            IF rtb_Divide_h >= 0.5 THEN 
                rtb_Add_d := rt_floorf(u := rtb_Add_d + 0.5);
            ELSE 
                rtb_Add_d := 0.0;
            END_IF;

        END_IF;

        (* Outputs for Atomic SubSystem: '<S676>/BatteryPackSignals' *)
        (* Product: '<S951>/Divide' incorporates:
         *  Constant: '<S811>/Constant8'
         *  SignalConversion: '<S682>/BusConversion_InsertedFor_IT_BatterySignal_Databus_at_inport_0' *)
        rtb_Add_en := rtb_Add_en / 100.0;
        (* End of Outputs for SubSystem: '<S676>/BatteryPackSignals' *)
        

        (* DataTypeConversion: '<S947>/Data Type Conversion2' *)
        rtb_Divide_h := ABS(rtb_Add_en);

        IF rtb_Divide_h < 8.388608E+6 THEN 

            IF rtb_Divide_h >= 0.5 THEN 
                rtb_Add_en := rt_floorf(u := rtb_Add_en + 0.5);
            ELSE 
                rtb_Add_en := 0.0;
            END_IF;

        END_IF;

        (* Outputs for Atomic SubSystem: '<S676>/BatteryPackSignals' *)
        (* Product: '<S964>/Divide' incorporates:
         *  Constant: '<S812>/Constant6'
         *  SignalConversion: '<S682>/BusConversion_InsertedFor_IT_BatterySignal_Databus_at_inport_0' *)
        rtb_Divide_h := rtb_Add_cw / 0.1;
        (* End of Outputs for SubSystem: '<S676>/BatteryPackSignals' *)
        

        (* DataTypeConversion: '<S960>/Data Type Conversion2' *)

        IF rtb_Divide_h >= 0.5 THEN 
            rtb_Add_ky := rt_floorf(u := rtb_Divide_h + 0.5);
        ELSE 
            rtb_Add_ky := 0.0;
        END_IF;

        (* Outputs for Atomic SubSystem: '<S676>/BatteryPackSignals' *)
        (* Product: '<S965>/Divide' incorporates:
         *  Constant: '<S812>/Constant8'
         *  SignalConversion: '<S682>/BusConversion_InsertedFor_IT_BatterySignal_Databus_at_inport_0' *)
        rtb_Divide_h := rtb_Add_bh / 0.1;
        (* End of Outputs for SubSystem: '<S676>/BatteryPackSignals' *)
        

        (* DataTypeConversion: '<S961>/Data Type Conversion2' *)

        IF rtb_Divide_h >= 0.5 THEN 
            rtb_Add_bh := rt_floorf(u := rtb_Divide_h + 0.5);
        ELSE 
            rtb_Add_bh := 0.0;
        END_IF;

        (* DataTypeConversion: '<S973>/Data Type Conversion4' *)
        v := ABS(rtb_BattSelect_i);

        IF v < 4.503599627370496E+15 THEN 

            IF v >= 0.5 THEN 
                rtb_BattSelect_i := rt_floord(u := rtb_BattSelect_i + 0.5);
            ELSE 
                rtb_BattSelect_i := 0.0;
            END_IF;

        END_IF;

        (* DataTypeConversion: '<S973>/Data Type Conversion1' *)
        v := ABS(rtb_BattSelect);

        IF v < 4.503599627370496E+15 THEN 

            IF v >= 0.5 THEN 
                rtb_BattSelect := rt_floord(u := rtb_BattSelect + 0.5);
            ELSE 
                rtb_BattSelect := 0.0;
            END_IF;

        END_IF;

        (* DataTypeConversion: '<S973>/Data Type Conversion3' *)
        v := ABS(rtb_BattSelect_f);

        IF v < 4.503599627370496E+15 THEN 

            IF v >= 0.5 THEN 
                rtb_BattSelect_f := rt_floord(u := rtb_BattSelect_f + 0.5);
            ELSE 
                rtb_BattSelect_f := 0.0;
            END_IF;

        END_IF;

        (* Outport: '<Root>/OP_ChiefMaster_IP_Msg1' incorporates:
         *  ArithShift: '<S973>/Shift Arithmetic1'
         *  ArithShift: '<S973>/Shift Arithmetic3'
         *  ArithShift: '<S973>/Shift Arithmetic5'
         *  ArithShift: '<S973>/Shift Arithmetic6'
         *  DataTypeConversion: '<S973>/Data Type Conversion1'
         *  DataTypeConversion: '<S973>/Data Type Conversion3'
         *  DataTypeConversion: '<S973>/Data Type Conversion4'
         *  DataTypeConversion: '<S973>/Data Type Conversion6'
         *  DataTypeConversion: '<S973>/Data Type Conversion7'
         *  SignalConversion: '<S677>/Signal Copy14'
         *  Sum: '<S973>/Add' *)
        OP_ChiefMaster_IP_Msg1[2] := UDINT_TO_USINT(USINT_TO_UDINT(UDINT_TO_USINT(USINT_TO_UDINT(UDINT_TO_USINT(USINT_TO_UDINT(UDINT_TO_USINT(USINT_TO_UDINT(UDINT_TO_USINT(USINT_TO_UDINT(UDINT_TO_USINT((DINT_TO_UDINT(DWORD_TO_DINT(SHL(DINT_TO_DWORD(BOOL_TO_DINT(DI_HVIL_Overrule)), 7))) + DINT_TO_UDINT(DWORD_TO_DINT(SHL(DINT_TO_DWORD(BOOL_TO_DINT(rtb_IT_boUDC_SafeToShutdown)), 6)))) + USINT_TO_UDINT(ShiftArithmetic4_m))) + USINT_TO_UDINT(BYTE_TO_USINT(SHL(USINT_TO_BYTE(DINT_TO_USINT(TRUNC(rtb_BattSelect_i))), 4))))) + USINT_TO_UDINT(ShiftArithmetic2_k))) + USINT_TO_UDINT(BYTE_TO_USINT(SHL(USINT_TO_BYTE(DINT_TO_USINT(TRUNC(rtb_BattSelect))), 2))))) + USINT_TO_UDINT(ShiftArithmetic_m))) + USINT_TO_UDINT(DINT_TO_USINT(TRUNC(rtb_BattSelect_f))));
        (* Product: '<S978>/Divide' incorporates:
         *  Constant: '<S976>/Constant2'
         *  Sum: '<S978>/Add' *)
        rtb_Divide_h := DINT_TO_REAL(rtb_Add_kr) / 0.1;
        (* DataTypeConversion: '<S977>/Data Type Conversion2' *)

        IF rtb_Divide_h >= 0.5 THEN 
            y_1 := rt_floorf(u := rtb_Divide_h + 0.5);
        ELSE 
            y_1 := 0.0;
        END_IF;

        (* DataTypeConversion: '<S981>/Data Type Conversion2' *)

        IF v_tmp < 4.503599627370496E+15 THEN 

            IF v_tmp >= 0.5 THEN 
                Count_k := rt_floord(u := REQ_HV_ON + 0.5);
            ELSE 
                Count_k := 0.0;
            END_IF;

        ELSE 
            Count_k := REQ_HV_ON;
        END_IF;

        (* DataTypeConversion: '<S981>/Data Type Conversion1' *)

        IF rtb_UnitDelay2 < 4.503599627370496E+15 THEN 

            IF rtb_UnitDelay2 >= 0.5 THEN 
                y := rt_floord(u := REQ_HV_ON_d + 0.5);
            ELSE 
                y := 0.0;
            END_IF;

        ELSE 
            y := REQ_HV_ON_d;
        END_IF;

        (* DataTypeConversion: '<S981>/Data Type Conversion' *)

        IF rtb_Uk1 < 4.503599627370496E+15 THEN 

            IF rtb_Uk1 >= 0.5 THEN 
                v := rt_floord(u := REQ_HV_ON_a + 0.5);
            ELSE 
                v := 0.0;
            END_IF;

        ELSE 
            v := REQ_HV_ON_a;
        END_IF;

        (* Outport: '<Root>/OP_ChiefMaster_OP_Msg2' incorporates:
         *  ArithShift: '<S981>/Shift Arithmetic'
         *  ArithShift: '<S981>/Shift Arithmetic1'
         *  ArithShift: '<S981>/Shift Arithmetic2'
         *  ArithShift: '<S981>/Shift Arithmetic3'
         *  ArithShift: '<S981>/Shift Arithmetic4'
         *  ArithShift: '<S982>/Shift Arithmetic'
         *  ArithShift: '<S982>/Shift Arithmetic1'
         *  DataTypeConversion: '<S981>/Data Type Conversion'
         *  DataTypeConversion: '<S981>/Data Type Conversion1'
         *  DataTypeConversion: '<S981>/Data Type Conversion2'
         *  DataTypeConversion: '<S981>/Data Type Conversion3'
         *  DataTypeConversion: '<S981>/Data Type Conversion4'
         *  DataTypeConversion: '<S981>/Data Type Conversion5'
         *  DataTypeConversion: '<S982>/Data Type Conversion'
         *  DataTypeConversion: '<S982>/Data Type Conversion1'
         *  DataTypeConversion: '<S982>/Data Type Conversion3'
         *  Outport: '<Root>/DO_boEMSRET_BB1_1'
         *  Sum: '<S981>/Add'
         *  Sum: '<S982>/Add' *)
        OP_ChiefMaster_OP_Msg2[1] := UDINT_TO_USINT(USINT_TO_UDINT(UDINT_TO_USINT(USINT_TO_UDINT(UDINT_TO_USINT(USINT_TO_UDINT(UDINT_TO_USINT(USINT_TO_UDINT(UDINT_TO_USINT(USINT_TO_UDINT(UDINT_TO_USINT(USINT_TO_UDINT(UDINT_TO_USINT(USINT_TO_UDINT(ShiftArithmetic6_i) + USINT_TO_UDINT(ShiftArithmetic5_k))) + DINT_TO_UDINT(DWORD_TO_DINT(SHL(DINT_TO_DWORD(BOOL_TO_DINT(DO_REQ_DC_ON_PLUS)), 5))))) + DINT_TO_UDINT(DWORD_TO_DINT(SHL(DINT_TO_DWORD(BOOL_TO_DINT(DO_REQ_DC_ON_MINUS)), 4))))) + USINT_TO_UDINT(BYTE_TO_USINT(SHL(USINT_TO_BYTE(DINT_TO_USINT(TRUNC(Count_k))), 3))))) + USINT_TO_UDINT(BYTE_TO_USINT(SHL(USINT_TO_BYTE(DINT_TO_USINT(TRUNC(y))), 2))))) + USINT_TO_UDINT(BYTE_TO_USINT(SHL(USINT_TO_BYTE(DINT_TO_USINT(TRUNC(v))), 1))))) + BOOL_TO_UDINT(DO_boKL15_IMD_BB3));
        OP_ChiefMaster_OP_Msg2[2] := UDINT_TO_USINT(USINT_TO_UDINT(UDINT_TO_USINT(USINT_TO_UDINT(UDINT_TO_USINT(USINT_TO_UDINT(UDINT_TO_USINT(USINT_TO_UDINT(UDINT_TO_USINT(USINT_TO_UDINT(UDINT_TO_USINT(USINT_TO_UDINT(UDINT_TO_USINT(USINT_TO_UDINT(ShiftArithmetic6_m) + USINT_TO_UDINT(ShiftArithmetic5_a))) + USINT_TO_UDINT(ShiftArithmetic4_a))) + USINT_TO_UDINT(ShiftArithmetic3_k))) + USINT_TO_UDINT(ShiftArithmetic2_p))) + DINT_TO_UDINT(DWORD_TO_DINT(SHL(DINT_TO_DWORD(BOOL_TO_DINT(DO_boResetButton_LED)), 2))))) + DINT_TO_UDINT(DWORD_TO_DINT(SHL(DINT_TO_DWORD(BOOL_TO_DINT(DO_boEMSRET_BB1_1)), 1))))) + BOOL_TO_UDINT(DO_CabinAlarm));
        (* ArithShift: '<S990>/Shift Arithmetic3' incorporates:
         *  DataTypeConversion: '<S990>/Data Type Conversion4' *)
        rtb_ShiftArithmetic3_p := DINT_TO_USINT(DWORD_TO_DINT(SHL(DINT_TO_DWORD(BOOL_TO_DINT(System_Error)), 4)));
        (* Outport: '<Root>/OP_ChiefMaster_SS1_Msg3' incorporates:
         *  ArithShift: '<S991>/Shift Arithmetic'
         *  ArithShift: '<S991>/Shift Arithmetic1'
         *  ArithShift: '<S991>/Shift Arithmetic3'
         *  ArithShift: '<S991>/Shift Arithmetic5'
         *  DataTypeConversion: '<S984>/Extract Desired Bits'
         *  DataTypeConversion: '<S985>/Extract Desired Bits'
         *  DataTypeConversion: '<S991>/Data Type Conversion'
         *  DataTypeConversion: '<S991>/Data Type Conversion3'
         *  Sum: '<S991>/Add' *)
        OP_ChiefMaster_SS1_Msg3[1] := UDINT_TO_USINT(USINT_TO_UDINT(UDINT_TO_USINT(USINT_TO_UDINT(UDINT_TO_USINT(USINT_TO_UDINT(UDINT_TO_USINT(USINT_TO_UDINT(UDINT_TO_USINT(USINT_TO_UDINT(UDINT_TO_USINT(USINT_TO_UDINT(UDINT_TO_USINT(DINT_TO_UDINT(DWORD_TO_DINT(SHL(DINT_TO_DWORD(USINT_TO_DINT(rtb_Out)) AND 3, 6))) + USINT_TO_UDINT(ShiftArithmetic6_h))) + USINT_TO_UDINT(ShiftArithmetic4_n))) + DINT_TO_UDINT(DWORD_TO_DINT(SHL(DINT_TO_DWORD(USINT_TO_DINT(rtb_ExtractDesiredBits_bk_tmp)), 4))))) + USINT_TO_UDINT(ShiftArithmetic2_d))) + DINT_TO_UDINT(DWORD_TO_DINT(SHL(DINT_TO_DWORD(USINT_TO_DINT(rtb_ExtractDesiredBits_b13)), 2))))) + DINT_TO_UDINT(DWORD_TO_DINT(SHL(DINT_TO_DWORD(BOOL_TO_DINT(rtb_IT_boBMS_HV_ON_BB)), 1))))) + BOOL_TO_UDINT(rtb_FL_boKL15_Reset));
        (* Outputs for Atomic SubSystem: '<S676>/BatteryPackSignals' *)
        (* Switch: '<S995>/Switch' incorporates:
         *  Constant: '<S994>/Constant2'
         *  SignalConversion: '<S682>/BusConversion_InsertedFor_IT_BatterySignal_Databus_at_inport_0' *)

        IF rtb_IP_boBMS_HV_REL_ON_BB1 THEN 
            rtb_Divide_h := rtb_Add_nm;
        ELSE 
            rtb_Divide_h := FL_sHVC_CellBalanceVoltage_mV;
        END_IF;

        (* End of Switch: '<S995>/Switch' *)
        (* End of Outputs for SubSystem: '<S676>/BatteryPackSignals' *)
        

        (* RelationalOperator: '<S996>/Relational Operator' incorporates:
         *  Constant: '<S994>/Constant2' *)
        rtb_boData_Out := rtb_Divide_h >= FL_sHVC_CellBalanceVoltage_mV;
        (* Outputs for Atomic SubSystem: '<S676>/BatteryPackSignals' *)
        (* Switch: '<S995>/Switch1' incorporates:
         *  Constant: '<S994>/Constant2'
         *  SignalConversion: '<S682>/BusConversion_InsertedFor_IT_BatterySignal_Databus_at_inport_0' *)

        IF rtb_IP_boBMS_HV_REL_ON_BB2 THEN 
            rtb_Divide_h := rtb_Add_d4;
        ELSE 
            rtb_Divide_h := FL_sHVC_CellBalanceVoltage_mV;
        END_IF;

        (* End of Switch: '<S995>/Switch1' *)
        (* End of Outputs for SubSystem: '<S676>/BatteryPackSignals' *)
        

        (* RelationalOperator: '<S996>/Relational Operator1' incorporates:
         *  Constant: '<S994>/Constant2' *)
        rtb_IT_boBMS_HV_ON_BB := rtb_Divide_h >= FL_sHVC_CellBalanceVoltage_mV;
        (* Outputs for Atomic SubSystem: '<S676>/BatteryPackSignals' *)
        (* Switch: '<S995>/Switch2' incorporates:
         *  Constant: '<S994>/Constant2'
         *  SignalConversion: '<S682>/BusConversion_InsertedFor_IT_BatterySignal_Databus_at_inport_0' *)

        IF rtb_IP_boBMS_HV_REL_ON_BB3 THEN 
            rtb_Divide_h := rtb_Add_cw;
        ELSE 
            rtb_Divide_h := FL_sHVC_CellBalanceVoltage_mV;
        END_IF;

        (* End of Switch: '<S995>/Switch2' *)
        (* End of Outputs for SubSystem: '<S676>/BatteryPackSignals' *)
        

        (* Outport: '<Root>/OP_ChiefMaster_SS1_Msg3' incorporates:
         *  ArithShift: '<S992>/Shift Arithmetic'
         *  ArithShift: '<S992>/Shift Arithmetic1'
         *  ArithShift: '<S992>/Shift Arithmetic4'
         *  ArithShift: '<S993>/Shift Arithmetic2'
         *  Constant: '<S994>/Constant2'
         *  DataTypeConversion: '<S987>/Extract Desired Bits'
         *  DataTypeConversion: '<S988>/Extract Desired Bits'
         *  DataTypeConversion: '<S989>/Extract Desired Bits'
         *  DataTypeConversion: '<S992>/Data Type Conversion'
         *  DataTypeConversion: '<S992>/Data Type Conversion1'
         *  DataTypeConversion: '<S992>/Data Type Conversion3'
         *  Logic: '<S996>/OR'
         *  RelationalOperator: '<S996>/Relational Operator2'
         *  Sum: '<S992>/Add'
         *  Sum: '<S993>/Add' *)
        OP_ChiefMaster_SS1_Msg3[2] := UDINT_TO_USINT(USINT_TO_UDINT(UDINT_TO_USINT(USINT_TO_UDINT(UDINT_TO_USINT(USINT_TO_UDINT(UDINT_TO_USINT(USINT_TO_UDINT(UDINT_TO_USINT(USINT_TO_UDINT(UDINT_TO_USINT(DINT_TO_UDINT(DWORD_TO_DINT(SHL(DINT_TO_DWORD(USINT_TO_DINT(rtb_IMD_State_g)) AND 7, 5))) + USINT_TO_UDINT(UDINT_TO_USINT(USINT_TO_UDINT(ShiftArithmetic6_n) + USINT_TO_UDINT(ShiftArithmetic5_a2))))) + USINT_TO_UDINT(ShiftArithmetic3_o))) + USINT_TO_UDINT(ShiftArithmetic2_b))) + DINT_TO_UDINT(DWORD_TO_DINT(SHL(DINT_TO_DWORD(BOOL_TO_DINT((rtb_boData_Out AND rtb_IT_boBMS_HV_ON_BB) AND (rtb_Divide_h >= FL_sHVC_CellBalanceVoltage_mV))), 2))))) + DINT_TO_UDINT(DWORD_TO_DINT(SHL(DINT_TO_DWORD(BOOL_TO_DINT(rtb_FL_boSS_HVIL_NOK)), 1))))) + BOOL_TO_UDINT(rtb_FL_boCMSleep));
        OP_ChiefMaster_SS1_Msg3[7] := UDINT_TO_USINT(USINT_TO_UDINT(UDINT_TO_USINT(USINT_TO_UDINT(UDINT_TO_USINT(USINT_TO_UDINT(UDINT_TO_USINT(USINT_TO_UDINT(UDINT_TO_USINT(USINT_TO_UDINT(UDINT_TO_USINT(USINT_TO_UDINT(UDINT_TO_USINT(USINT_TO_UDINT(ShiftArithmetic6_k) + USINT_TO_UDINT(ShiftArithmetic5_i))) + USINT_TO_UDINT(ShiftArithmetic4_ap))) + USINT_TO_UDINT(ShiftArithmetic3_e))) + DINT_TO_UDINT(DWORD_TO_DINT(SHL(DINT_TO_DWORD(USINT_TO_DINT(rtb_IMD_State)) AND 7, 3))))) + USINT_TO_UDINT(ShiftArithmetic1))) + USINT_TO_UDINT(ShiftArithmetic_h))) + DINT_TO_UDINT(DWORD_TO_DINT(DINT_TO_DWORD(USINT_TO_DINT(rtb_System_SD_ErrorCode)) AND 7)));
        (* Outputs for Atomic SubSystem: '<S676>/BatteryPackSignals' *)
        (* Product: '<S1002>/Divide' incorporates:
         *  Constant: '<S997>/Constant1'
         *  SignalConversion: '<S682>/BusConversion_InsertedFor_IT_BatterySignal_Databus_at_inport_0'
         *  Sum: '<S119>/Add' *)
        rtb_Divide_h := ((rtb_Add_ki5 + rtb_Add_ir) + rtb_Add_m) / 0.1;
        (* End of Outputs for SubSystem: '<S676>/BatteryPackSignals' *)
        

        (* DataTypeConversion: '<S1001>/Data Type Conversion2' *)

        IF ABS(rtb_Divide_h) >= 0.5 THEN 
            rtb_Add_nm := rt_floorf(u := rtb_Divide_h + 0.5);
        ELSE 
            rtb_Add_nm := 0.0;
        END_IF;

        (* DataTypeConversion: '<S1005>/Data Type Conversion2' incorporates:
         *  MinMax: '<S120>/Min' *)

        IF maxV >= 0.5 THEN 
            maxV := rt_floorf(u := maxV + 0.5);
        ELSE 
            maxV := 0.0;
        END_IF;

        (* DataTypeConversion: '<S1009>/Data Type Conversion2' incorporates:
         *  Sum: '<S1010>/Add' *)
        rtb_Divide_h := ABS(FL_sST_MaxChargeCurrent);

        IF rtb_Divide_h < 8.388608E+6 THEN 

            IF rtb_Divide_h >= 0.5 THEN 
                rtb_Add_d4 := rt_floorf(u := FL_sST_MaxChargeCurrent + 0.5);
            ELSE 
                rtb_Add_d4 := 0.0;
            END_IF;

        ELSE 
            rtb_Add_d4 := FL_sST_MaxChargeCurrent;
        END_IF;

        (* DataTypeConversion: '<S1013>/Data Type Conversion2' incorporates:
         *  Sum: '<S1014>/Add' *)
        rtb_Divide_h := ABS(rtb_FL_sSS_MaxDisChargeCurrent);

        IF rtb_Divide_h < 8.388608E+6 THEN 

            IF rtb_Divide_h >= 0.5 THEN 
                rtb_FL_sSS_MaxDisChargeCurrent := rt_floorf(u := rtb_FL_sSS_MaxDisChargeCurrent + 0.5);
            ELSE 
                rtb_FL_sSS_MaxDisChargeCurrent := 0.0;
            END_IF;

        END_IF;

        (* DataTypeConversion: '<S1020>/Data Type Conversion3' *)

        IF rtb_Uk1 < 4.503599627370496E+15 THEN 

            IF rtb_Uk1 >= 0.5 THEN 
                Count_k := rt_floord(u := REQ_HV_ON_a + 0.5);
            ELSE 
                Count_k := 0.0;
            END_IF;

        ELSE 
            Count_k := REQ_HV_ON_a;
        END_IF;

        (* Outport: '<Root>/BMS_Control_Batt1' incorporates:
         *  DataTypeConversion: '<S1020>/Data Type Conversion3'
         *  Sum: '<S1020>/Add' *)
        BMS_Control_Batt1[0] := UDINT_TO_USINT(USINT_TO_UDINT(UDINT_TO_USINT(USINT_TO_UDINT(UDINT_TO_USINT(USINT_TO_UDINT(UDINT_TO_USINT(USINT_TO_UDINT(UDINT_TO_USINT(USINT_TO_UDINT(UDINT_TO_USINT(USINT_TO_UDINT(UDINT_TO_USINT(USINT_TO_UDINT(ShiftArithmetic6_kx) + USINT_TO_UDINT(ShiftArithmetic5_ke))) + USINT_TO_UDINT(ShiftArithmetic4_d))) + USINT_TO_UDINT(ShiftArithmetic3_oe))) + USINT_TO_UDINT(ShiftArithmetic2_ot))) + USINT_TO_UDINT(ShiftArithmetic1_n))) + OP_ChiefMaster_Battery1_Msg7_tmp)) + USINT_TO_UDINT(DINT_TO_USINT(TRUNC(Count_k))));
        (* DataTypeConversion: '<S1021>/Data Type Conversion3' *)

        IF rtb_UnitDelay2 < 4.503599627370496E+15 THEN 

            IF rtb_UnitDelay2 >= 0.5 THEN 
                Count_k := rt_floord(u := REQ_HV_ON_d + 0.5);
            ELSE 
                Count_k := 0.0;
            END_IF;

        ELSE 
            Count_k := REQ_HV_ON_d;
        END_IF;

        (* Outport: '<Root>/BMS_Control_Batt2' incorporates:
         *  DataTypeConversion: '<S1021>/Data Type Conversion3'
         *  Sum: '<S1021>/Add' *)
        BMS_Control_Batt2[0] := UDINT_TO_USINT(USINT_TO_UDINT(UDINT_TO_USINT(USINT_TO_UDINT(UDINT_TO_USINT(USINT_TO_UDINT(UDINT_TO_USINT(USINT_TO_UDINT(UDINT_TO_USINT(USINT_TO_UDINT(UDINT_TO_USINT(USINT_TO_UDINT(UDINT_TO_USINT(USINT_TO_UDINT(ShiftArithmetic6_kxt) + USINT_TO_UDINT(ShiftArithmetic5_hi))) + USINT_TO_UDINT(ShiftArithmetic4_b))) + USINT_TO_UDINT(ShiftArithmetic3_o0))) + USINT_TO_UDINT(ShiftArithmetic2_e))) + USINT_TO_UDINT(ShiftArithmetic1_nm))) + OP_ChiefMaster_Battery2_Msg10_tmp)) + USINT_TO_UDINT(DINT_TO_USINT(TRUNC(Count_k))));
        (* DataTypeConversion: '<S1022>/Data Type Conversion3' *)

        IF v_tmp < 4.503599627370496E+15 THEN 

            IF v_tmp >= 0.5 THEN 
                Count_k := rt_floord(u := REQ_HV_ON + 0.5);
            ELSE 
                Count_k := 0.0;
            END_IF;

        ELSE 
            Count_k := REQ_HV_ON;
        END_IF;

        (* Outport: '<Root>/BMS_Control_Batt3' incorporates:
         *  DataTypeConversion: '<S1022>/Data Type Conversion3'
         *  Sum: '<S1022>/Add' *)
        BMS_Control_Batt3[0] := UDINT_TO_USINT(USINT_TO_UDINT(UDINT_TO_USINT(USINT_TO_UDINT(UDINT_TO_USINT(USINT_TO_UDINT(UDINT_TO_USINT(USINT_TO_UDINT(UDINT_TO_USINT(USINT_TO_UDINT(UDINT_TO_USINT(USINT_TO_UDINT(UDINT_TO_USINT(USINT_TO_UDINT(ShiftArithmetic6_b) + USINT_TO_UDINT(ShiftArithmetic5_b))) + USINT_TO_UDINT(ShiftArithmetic4_p))) + USINT_TO_UDINT(ShiftArithmetic3_a))) + USINT_TO_UDINT(ShiftArithmetic2_m))) + USINT_TO_UDINT(ShiftArithmetic1_nx))) + OP_ChiefMaster_Battery3_Msg13_tmp)) + USINT_TO_UDINT(DINT_TO_USINT(TRUNC(Count_k))));
        (* DataTypeConversion: '<S1031>/Data Type Conversion1' *)

        IF rtb_Uk1 < 4.503599627370496E+15 THEN 

            IF rtb_Uk1 >= 0.5 THEN 
                Count_k := rt_floord(u := REQ_HV_ON_a + 0.5);
            ELSE 
                Count_k := 0.0;
            END_IF;

        ELSE 
            Count_k := REQ_HV_ON_a;
        END_IF;

        (* Outport: '<Root>/OP_LiBa_OperationRequest_Batt1' incorporates:
         *  ArithShift: '<S1031>/Shift Arithmetic1'
         *  DataTypeConversion: '<S1031>/Data Type Conversion1'
         *  Sum: '<S1031>/Add' *)
        OP_LiBa_OperationRequest_Batt1[0] := UDINT_TO_USINT(USINT_TO_UDINT(UDINT_TO_USINT(USINT_TO_UDINT(UDINT_TO_USINT(USINT_TO_UDINT(UDINT_TO_USINT(USINT_TO_UDINT(UDINT_TO_USINT(USINT_TO_UDINT(UDINT_TO_USINT(USINT_TO_UDINT(UDINT_TO_USINT(USINT_TO_UDINT(ShiftArithmetic6_ap) + USINT_TO_UDINT(ShiftArithmetic5_m))) + USINT_TO_UDINT(ShiftArithmetic4_l))) + USINT_TO_UDINT(ShiftArithmetic3_h))) + USINT_TO_UDINT(ShiftArithmetic2_f))) + USINT_TO_UDINT(BYTE_TO_USINT(SHL(USINT_TO_BYTE(DINT_TO_USINT(TRUNC(Count_k))), 2))))) + USINT_TO_UDINT(ShiftArithmetic_k))) + USINT_TO_UDINT(DataTypeConversion3));
        (* DataTypeConversion: '<S1037>/Data Type Conversion1' *)

        IF rtb_UnitDelay2 < 4.503599627370496E+15 THEN 

            IF rtb_UnitDelay2 >= 0.5 THEN 
                Count_k := rt_floord(u := REQ_HV_ON_d + 0.5);
            ELSE 
                Count_k := 0.0;
            END_IF;

        ELSE 
            Count_k := REQ_HV_ON_d;
        END_IF;

        (* Outport: '<Root>/OP_LiBa_OperationRequest_Batt2' incorporates:
         *  ArithShift: '<S1037>/Shift Arithmetic1'
         *  DataTypeConversion: '<S1037>/Data Type Conversion1'
         *  Sum: '<S1037>/Add' *)
        OP_LiBa_OperationRequest_Batt2[0] := UDINT_TO_USINT(USINT_TO_UDINT(UDINT_TO_USINT(USINT_TO_UDINT(UDINT_TO_USINT(USINT_TO_UDINT(UDINT_TO_USINT(USINT_TO_UDINT(UDINT_TO_USINT(USINT_TO_UDINT(UDINT_TO_USINT(USINT_TO_UDINT(UDINT_TO_USINT(USINT_TO_UDINT(ShiftArithmetic6_o) + USINT_TO_UDINT(ShiftArithmetic5_k0))) + USINT_TO_UDINT(ShiftArithmetic4_f))) + USINT_TO_UDINT(ShiftArithmetic3_l))) + USINT_TO_UDINT(ShiftArithmetic2_fl))) + USINT_TO_UDINT(BYTE_TO_USINT(SHL(USINT_TO_BYTE(DINT_TO_USINT(TRUNC(Count_k))), 2))))) + USINT_TO_UDINT(ShiftArithmetic_a))) + USINT_TO_UDINT(DataTypeConversion3_d));
        (* DataTypeConversion: '<S1043>/Data Type Conversion1' *)

        IF v_tmp < 4.503599627370496E+15 THEN 

            IF v_tmp >= 0.5 THEN 
                Count_k := rt_floord(u := REQ_HV_ON + 0.5);
            ELSE 
                Count_k := 0.0;
            END_IF;

        ELSE 
            Count_k := REQ_HV_ON;
        END_IF;

        (* Outport: '<Root>/OP_LiBa_OperationRequest_Batt3' incorporates:
         *  ArithShift: '<S1043>/Shift Arithmetic1'
         *  DataTypeConversion: '<S1043>/Data Type Conversion1'
         *  Sum: '<S1043>/Add' *)
        OP_LiBa_OperationRequest_Batt3[0] := UDINT_TO_USINT(USINT_TO_UDINT(UDINT_TO_USINT(USINT_TO_UDINT(UDINT_TO_USINT(USINT_TO_UDINT(UDINT_TO_USINT(USINT_TO_UDINT(UDINT_TO_USINT(USINT_TO_UDINT(UDINT_TO_USINT(USINT_TO_UDINT(UDINT_TO_USINT(USINT_TO_UDINT(ShiftArithmetic6_mw) + USINT_TO_UDINT(ShiftArithmetic5_c))) + USINT_TO_UDINT(ShiftArithmetic4_db))) + USINT_TO_UDINT(ShiftArithmetic3_c))) + USINT_TO_UDINT(ShiftArithmetic2_g))) + USINT_TO_UDINT(BYTE_TO_USINT(SHL(USINT_TO_BYTE(DINT_TO_USINT(TRUNC(Count_k))), 2))))) + USINT_TO_UDINT(ShiftArithmetic_p))) + USINT_TO_UDINT(DataTypeConversion3_l));
        (* Update for UnitDelay: '<S10>/Unit Delay' *)
        UnitDelay_DSTATE := 0.0;
        (* Update for UnitDelay: '<S10>/Unit Delay6' *)
        UnitDelay6_DSTATE := rtb_Contactor_FB_State_h;
        (* Update for UnitDelay: '<S10>/Unit Delay1' *)
        UnitDelay1_DSTATE := 0.0;
        (* Update for UnitDelay: '<S10>/Unit Delay7' *)
        UnitDelay7_DSTATE := rtb_Contactor_FB_State_g;
        (* Update for UnitDelay: '<S10>/Unit Delay2' *)
        UnitDelay2_DSTATE := 0.0;
        (* Update for UnitDelay: '<S10>/Unit Delay8' *)
        UnitDelay8_DSTATE := rtb_Contactor_FB_State;
        (* Update for Delay: '<S768>/Delay' *)
        Delay_DSTATE[0] := Delay_DSTATE[1];
        (* Update for Delay: '<S766>/Delay' *)
        Delay_DSTATE_o[0] := Delay_DSTATE_o[1];
        (* Update for Delay: '<S767>/Delay' *)
        Delay_DSTATE_k[0] := Delay_DSTATE_k[1];
        (* Update for Delay: '<S723>/Delay' *)
        Delay_DSTATE_a[0] := Delay_DSTATE_a[1];
        (* Update for Delay: '<S721>/Delay' *)
        Delay_DSTATE_ov[0] := Delay_DSTATE_ov[1];
        (* Update for Delay: '<S722>/Delay' *)
        Delay_DSTATE_c[0] := Delay_DSTATE_c[1];
        (* Update for Delay: '<S768>/Delay' *)
        Delay_DSTATE[1] := Delay_DSTATE[2];
        (* Update for Delay: '<S766>/Delay' *)
        Delay_DSTATE_o[1] := Delay_DSTATE_o[2];
        (* Update for Delay: '<S767>/Delay' *)
        Delay_DSTATE_k[1] := Delay_DSTATE_k[2];
        (* Update for Delay: '<S723>/Delay' *)
        Delay_DSTATE_a[1] := Delay_DSTATE_a[2];
        (* Update for Delay: '<S721>/Delay' *)
        Delay_DSTATE_ov[1] := Delay_DSTATE_ov[2];
        (* Update for Delay: '<S722>/Delay' *)
        Delay_DSTATE_c[1] := Delay_DSTATE_c[2];
        (* Update for Delay: '<S768>/Delay' *)
        Delay_DSTATE[2] := rtb_IT_boChargeStop_Button;
        (* Update for Delay: '<S766>/Delay' *)
        Delay_DSTATE_o[2] := rtb_IT_boChargeStop_Button;
        (* Update for Delay: '<S767>/Delay' *)
        Delay_DSTATE_k[2] := rtb_IT_boChargeStop_Button;
        (* Update for Delay: '<S723>/Delay' *)
        Delay_DSTATE_a[2] := rtb_IT_boChargeStop_Button;
        (* Update for Delay: '<S721>/Delay' *)
        Delay_DSTATE_ov[2] := rtb_UnitDelay1_d;
        (* Update for Delay: '<S722>/Delay' *)
        Delay_DSTATE_c[2] := rtb_Out_bl;
        (* Update for UnitDelay: '<S8>/Unit Delay5' *)
        UnitDelay5_DSTATE := 0.0;
        (* Update for UnitDelay: '<S8>/Unit Delay4' *)
        UnitDelay4_DSTATE := 0.0;
        (* Update for UnitDelay: '<S8>/Unit Delay3' *)
        UnitDelay3_DSTATE := 0.0;
        (* Update for UnitDelay: '<S8>/Unit Delay2' *)
        UnitDelay2_DSTATE_d := REQ_HV_Open_Batt1;
        (* Update for UnitDelay: '<S8>/Unit Delay6' *)
        UnitDelay6_DSTATE_b := REQ_HV_Open_Batt2;
        (* Update for UnitDelay: '<S8>/Unit Delay7' *)
        UnitDelay7_DSTATE_j := REQ_HV_Open_Batt3;
        (* Update for UnitDelay: '<S8>/Unit Delay9' *)
        UnitDelay9_DSTATE := System_Error;
        (* Update for UnitDelay: '<S8>/Unit Delay1' *)
        UnitDelay1_DSTATE_fl := rtb_Delay_j;
        (* Update for UnitDelay: '<S35>/Unit Delay1' *)
        UnitDelay1_DSTATE_f := MainHV_Minus_Status;
        (* Update for UnitDelay: '<S35>/Unit Delay' *)
        UnitDelay_DSTATE_o := MainHV_Plus_Status;
        (* Update for UnitDelay: '<S35>/Unit Delay2' *)
        UnitDelay2_DSTATE_g := rtb_Out_k;
        (* Update for UnitDelay: '<S13>/Unit Delay3' *)
        UnitDelay3_DSTATE_p := MainHV_Plus_Status;
        (* Update for UnitDelay: '<S13>/Unit Delay2' *)
        UnitDelay2_DSTATE_a := MainHV_Minus_Status;
        (* Update for UnitDelay: '<S13>/Unit Delay6' *)
        UnitDelay6_DSTATE_h := System_Error;
        (* Update for UnitDelay: '<S13>/Unit Delay5' *)
        UnitDelay5_DSTATE_e := MainHV_Minus_Status;
        (* Update for UnitDelay: '<S13>/Unit Delay1' *)
        UnitDelay1_DSTATE_b := System_Error;
        (* Update for UnitDelay: '<S110>/Unit Delay' *)
        UnitDelay_DSTATE_h := FL_sST_MaxChargeCurrent;
        (* Outputs for Atomic SubSystem: '<S676>/BatteryPackSignals' *)
        (* Update for UnitDelay: '<S121>/Unit Delay' incorporates:
         *  SignalConversion: '<S698>/Signal Copy' *)
        UnitDelay_DSTATE_d := rtb_IP_boBMS_SDError_BB1;
        (* Update for UnitDelay: '<S121>/Unit Delay1' incorporates:
         *  SignalConversion: '<S699>/Signal Copy' *)
        UnitDelay1_DSTATE_m := rtb_IP_boBMS_SDError_BB2;
        (* Update for UnitDelay: '<S121>/Unit Delay2' incorporates:
         *  SignalConversion: '<S700>/Signal Copy' *)
        UnitDelay2_DSTATE_m := rtb_IP_boBMS_SDError_BB3;
        (* Outport: '<Root>/OP_ChiefMaster_SS1_Msg3' incorporates:
         *  SignalConversion: '<S677>/Signal Copy10'
         *  SignalConversion: '<S677>/Signal Copy11'
         *  SignalConversion: '<S677>/Signal Copy9'
         *  SignalConversion: '<S682>/BusConversion_InsertedFor_IT_BatterySignal_Databus_at_inport_0'
         *  SignalConversion: '<S698>/Signal Copy'
         *  SignalConversion: '<S699>/Signal Copy'
         *  SignalConversion: '<S700>/Signal Copy' *)
        i0_SDError(ssMethodType := SS_UPDATE, FL_boKL15_Reset := rtb_FL_boKL15_Reset, IT_Databus := rtb_ExtractDesiredBits_b13, IT_Databus_m := rtb_IP_boBMS_HV_REL_ON_BB1, IT_Databus_n := rtb_IP_boBMS_SDError_BB1, IT_Databus_a := rtb_IP_boBMS_HV_REL_ON_BB2, IT_Databus_o := rtb_IP_boBMS_SDError_BB2, IT_Databus_or := rtb_IP_boBMS_HV_REL_ON_BB3, IT_Databus_i := rtb_IP_boBMS_SDError_BB3, IT_Databus_c := rtb_Add_ki5, IT_Databus_o3 := rtb_Add_ir, IT_Databus_e := rtb_Add_m, IT_Databus_n0 := rtb_IT_boHW_HVIL_BDU, IT_Databus_ep := rtb_out_i, IT_Databus_l := rtb_out_ne, IT_Databus_f := rtb_IP_boBMS_IMD_Active_BB1, IT_Databus_k := rtb_IP_boBMS_IMD_Active_BB2, IT_Databus_g := rtb_IP_boBMS_IMD_Active_BB3, IT_Databus_b := rtb_S_in, IT_Databus_d := rtb_AND_l2, IT_Databus_h := rtb_IP_boBatt1_Actia_Availability, IT_Databus_j := rtb_AND_ni, IT_Databus_ja := rtb_Delay_dl, IT_Databus_if := rtb_AND_ma, FL_BDUControl_Databus := MainHV_Minus_Status, FL_BDUControl_Databus_o := MainHV_Plus_Status, FL_BDUControl_Databus_n := Precharge_Satus, FL_BatteryBox_HVControl_Databus := REQ_HV_ON_a, FL_BatteryBox_HVControl_Databus_b := REQ_HV_ON_d, FL_BatteryBox_HVControl_Databus_a := REQ_HV_ON, FL_u8SS_EmergencySD := rtb_Delay_j);
        System_Error := i0_SDError.FL_boSS_System_SD;
        OP_ChiefMaster_SS1_Msg3[5] := i0_SDError.FL_u8SS_System_SD_ErrorCode;
        (* End of Outputs for SubSystem: '<S676>/BatteryPackSignals' *)
        

        (* Update for UnitDelay: '<S29>/Delay Input1' incorporates:
         *  Constant: '<S13>/Constant'
         *
         * Block description for '<S29>/Delay Input1':
         *  
         *  Store in Global RAM *)
        DelayInput1_DSTATE := 0.0;
        (* Update for UnitDelay: '<S21>/Unit Delay' *)
        UnitDelay_DSTATE_i := WeldingDetection_Status;
        (* Update for UnitDelay: '<S94>/Delay Input1' incorporates:
         *  Outport: '<Root>/DO_KL15_BB1'
         *  RelationalOperator: '<S95>/Compare'
         *
         * Block description for '<S94>/Delay Input1':
         *  
         *  Store in Global RAM *)
        DelayInput1_DSTATE_g := DO_KL15_BB1;
        (* Update for UnitDelay: '<S99>/Delay Input1' incorporates:
         *  Outport: '<Root>/DO_KL15_BB2'
         *  RelationalOperator: '<S100>/Compare'
         *
         * Block description for '<S99>/Delay Input1':
         *  
         *  Store in Global RAM *)
        DelayInput1_DSTATE_n := DO_KL15_BB2;
        (* Update for UnitDelay: '<S104>/Delay Input1' incorporates:
         *  Outport: '<Root>/DO_KL15_BB3'
         *  RelationalOperator: '<S105>/Compare'
         *
         * Block description for '<S104>/Delay Input1':
         *  
         *  Store in Global RAM *)
        DelayInput1_DSTATE_e := DO_KL15_BB3;
        (* Update for UnitDelay: '<S12>/Unit Delay4' *)
        UnitDelay4_DSTATE_n := DO_REQ_MainHV_ON_MINUS;
        (* Update for UnitDelay: '<S12>/Unit Delay1' *)
        UnitDelay1_DSTATE_l := MainHV_Plus_Status;
        (* Update for UnitDelay: '<S122>/Unit Delay9' *)
        UnitDelay9_DSTATE_d := rtb_IT_boChargeStop_Button;
        (* Update for UnitDelay: '<S122>/Unit Delay8' *)
        UnitDelay8_DSTATE_k := rtb_UnitDelay1_d;
        (* Update for UnitDelay: '<S122>/Unit Delay7' *)
        UnitDelay7_DSTATE_h := rtb_Out_bl;
        (* End of Outputs for SubSystem: '<Root>/ChiefMaster' *)
        

        (* Outport: '<Root>/CMSleep' *)
        CMSleep := rtb_FL_boCMSleep;
        (* Outport: '<Root>/DO_boEMSRET_BDU1' incorporates:
         *  Outport: '<Root>/DO_boEMSRET_BB1_1' *)
        DO_boEMSRET_BDU1 := DO_boEMSRET_BB1_1;
        (* Outport: '<Root>/DO_boEMSRET_BDU2' incorporates:
         *  Outport: '<Root>/DO_boEMSRET_BB1_1' *)
        DO_boEMSRET_BDU2 := DO_boEMSRET_BB1_1;
        (* Outport: '<Root>/DO_boEMSRET_BB1_2' incorporates:
         *  Outport: '<Root>/DO_boEMSRET_BB1_1' *)
        DO_boEMSRET_BB1_2 := DO_boEMSRET_BB1_1;
        (* Outport: '<Root>/DO_boEMSRET_BB2_1' incorporates:
         *  Outport: '<Root>/DO_boEMSRET_BB1_1' *)
        DO_boEMSRET_BB2_1 := DO_boEMSRET_BB1_1;
        (* Outport: '<Root>/DO_boEMSRET_BB2_2' incorporates:
         *  Outport: '<Root>/DO_boEMSRET_BB1_1' *)
        DO_boEMSRET_BB2_2 := DO_boEMSRET_BB1_1;
        (* Outport: '<Root>/DO_boEMSRET_BB3_1' incorporates:
         *  Outport: '<Root>/DO_boEMSRET_BB1_1' *)
        DO_boEMSRET_BB3_1 := DO_boEMSRET_BB1_1;
        (* Outport: '<Root>/DO_boEMSRET_BB3_2' incorporates:
         *  Outport: '<Root>/DO_boEMSRET_BB1_1' *)
        DO_boEMSRET_BB3_2 := DO_boEMSRET_BB1_1;
        (* Outport: '<Root>/DO_HVIL_Supply' incorporates:
         *  Constant: '<S801>/Constant' *)
        DO_HVIL_Supply := OP_boHVIL_Supply;
        (* Outport: '<Root>/BMS_Control_Batt1' incorporates:
         *  Constant: '<S1017>/Constant3' *)
        BMS_Control_Batt1[1] := 0;
        BMS_Control_Batt1[2] := 0;
        BMS_Control_Batt1[3] := 0;
        BMS_Control_Batt1[4] := 0;
        BMS_Control_Batt1[5] := 0;
        BMS_Control_Batt1[6] := 0;
        BMS_Control_Batt1[7] := 0;
        (* Outport: '<Root>/BMS_Control_Batt2' incorporates:
         *  Constant: '<S1018>/Constant4' *)
        BMS_Control_Batt2[1] := 0;
        BMS_Control_Batt2[2] := 0;
        BMS_Control_Batt2[3] := 0;
        BMS_Control_Batt2[4] := 0;
        BMS_Control_Batt2[5] := 0;
        BMS_Control_Batt2[6] := 0;
        BMS_Control_Batt2[7] := 0;
        (* Outport: '<Root>/BMS_Control_Batt3' incorporates:
         *  Constant: '<S1019>/Constant5' *)
        BMS_Control_Batt3[1] := 0;
        BMS_Control_Batt3[2] := 0;
        BMS_Control_Batt3[3] := 0;
        BMS_Control_Batt3[4] := 0;
        BMS_Control_Batt3[5] := 0;
        BMS_Control_Batt3[6] := 0;
        BMS_Control_Batt3[7] := 0;
        (* Outputs for Atomic SubSystem: '<Root>/ChiefMaster' *)
        (* Outport: '<Root>/OP_LiBa_OperationRequest_Batt1' incorporates:
         *  Constant: '<S1023>/Constant'
         *  DataTypeConversion: '<S1023>/Data Type Conversion2'
         *  DataTypeConversion: '<S1029>/Extract Desired Bits' *)
        OP_LiBa_OperationRequest_Batt1[1] := BOOL_TO_USINT(DO_boKL15_IMD_BB1);
        (* End of Outputs for SubSystem: '<Root>/ChiefMaster' *)
        OP_LiBa_OperationRequest_Batt1[2] := 0;
        OP_LiBa_OperationRequest_Batt1[3] := 0;
        OP_LiBa_OperationRequest_Batt1[4] := 0;
        OP_LiBa_OperationRequest_Batt1[5] := 0;
        OP_LiBa_OperationRequest_Batt1[6] := 0;
        OP_LiBa_OperationRequest_Batt1[7] := 0;
        (* Outputs for Atomic SubSystem: '<Root>/ChiefMaster' *)
        (* Outport: '<Root>/OP_LiBa_OperationRequest_Batt2' incorporates:
         *  Constant: '<S1024>/Constant'
         *  DataTypeConversion: '<S1024>/Data Type Conversion2'
         *  DataTypeConversion: '<S1035>/Extract Desired Bits' *)
        OP_LiBa_OperationRequest_Batt2[1] := BOOL_TO_USINT(DO_boKL15_IMD_BB2);
        (* End of Outputs for SubSystem: '<Root>/ChiefMaster' *)
        OP_LiBa_OperationRequest_Batt2[2] := 0;
        OP_LiBa_OperationRequest_Batt2[3] := 0;
        OP_LiBa_OperationRequest_Batt2[4] := 0;
        OP_LiBa_OperationRequest_Batt2[5] := 0;
        OP_LiBa_OperationRequest_Batt2[6] := 0;
        OP_LiBa_OperationRequest_Batt2[7] := 0;
        (* Outputs for Atomic SubSystem: '<Root>/ChiefMaster' *)
        (* Outport: '<Root>/OP_LiBa_OperationRequest_Batt3' incorporates:
         *  Constant: '<S1025>/Constant'
         *  DataTypeConversion: '<S1025>/Data Type Conversion2'
         *  DataTypeConversion: '<S1041>/Extract Desired Bits'
         *  DataTypeConversion: '<S1042>/Extract Desired Bits' *)
        OP_LiBa_OperationRequest_Batt3[1] := BOOL_TO_USINT(DO_boKL15_IMD_BB3);
        OP_LiBa_OperationRequest_Batt3[2] := 0;
        (* End of Outputs for SubSystem: '<Root>/ChiefMaster' *)
        OP_LiBa_OperationRequest_Batt3[3] := 0;
        OP_LiBa_OperationRequest_Batt3[4] := 0;
        OP_LiBa_OperationRequest_Batt3[5] := 0;
        OP_LiBa_OperationRequest_Batt3[6] := 0;
        OP_LiBa_OperationRequest_Batt3[7] := 0;
        (* Outputs for Atomic SubSystem: '<Root>/ChiefMaster' *)
        (* Outport: '<Root>/OP_ChiefMaster_IP_Msg1' incorporates:
         *  ArithShift: '<S974>/Shift Arithmetic'
         *  ArithShift: '<S974>/Shift Arithmetic1'
         *  ArithShift: '<S974>/Shift Arithmetic2'
         *  ArithShift: '<S974>/Shift Arithmetic3'
         *  ArithShift: '<S974>/Shift Arithmetic4'
         *  ArithShift: '<S974>/Shift Arithmetic5'
         *  ArithShift: '<S974>/Shift Arithmetic6'
         *  ArithShift: '<S975>/Shift Arithmetic'
         *  ArithShift: '<S975>/Shift Arithmetic1'
         *  ArithShift: '<S975>/Shift Arithmetic2'
         *  ArithShift: '<S975>/Shift Arithmetic3'
         *  ArithShift: '<S975>/Shift Arithmetic4'
         *  ArithShift: '<S975>/Shift Arithmetic5'
         *  ArithShift: '<S975>/Shift Arithmetic6'
         *  Constant: '<S813>/Constant1'
         *  DataTypeConversion: '<S974>/Data Type Conversion'
         *  DataTypeConversion: '<S974>/Data Type Conversion1'
         *  DataTypeConversion: '<S974>/Data Type Conversion2'
         *  DataTypeConversion: '<S974>/Data Type Conversion3'
         *  DataTypeConversion: '<S974>/Data Type Conversion4'
         *  DataTypeConversion: '<S974>/Data Type Conversion5'
         *  DataTypeConversion: '<S974>/Data Type Conversion6'
         *  DataTypeConversion: '<S974>/Data Type Conversion7'
         *  DataTypeConversion: '<S975>/Data Type Conversion'
         *  DataTypeConversion: '<S975>/Data Type Conversion1'
         *  DataTypeConversion: '<S975>/Data Type Conversion2'
         *  DataTypeConversion: '<S975>/Data Type Conversion3'
         *  DataTypeConversion: '<S975>/Data Type Conversion4'
         *  DataTypeConversion: '<S975>/Data Type Conversion5'
         *  DataTypeConversion: '<S975>/Data Type Conversion6'
         *  DataTypeConversion: '<S975>/Data Type Conversion7'
         *  DataTypeConversion: '<S977>/Data Type Conversion2'
         *  DataTypeConversion: '<S979>/Extract Desired Bits'
         *  DataTypeConversion: '<S980>/Extract Desired Bits'
         *  SignalConversion: '<S677>/Signal Copy1'
         *  SignalConversion: '<S677>/Signal Copy10'
         *  SignalConversion: '<S677>/Signal Copy11'
         *  SignalConversion: '<S677>/Signal Copy2'
         *  SignalConversion: '<S677>/Signal Copy3'
         *  SignalConversion: '<S677>/Signal Copy8'
         *  SignalConversion: '<S677>/Signal Copy9'
         *  Sum: '<S974>/Add'
         *  Sum: '<S975>/Add' *)
        OP_ChiefMaster_IP_Msg1[0] := UDINT_TO_USINT(((((((DINT_TO_UDINT(DWORD_TO_DINT(SHL(DINT_TO_DWORD(BOOL_TO_DINT(rtb_IT_boHW_MainHV_Minus_FB)), 7))) + DINT_TO_UDINT(DWORD_TO_DINT(SHL(DINT_TO_DWORD(BOOL_TO_DINT(rtb_IT_boHW_MainHV_Plus_FB)), 6)))) + DINT_TO_UDINT(DWORD_TO_DINT(SHL(DINT_TO_DWORD(BOOL_TO_DINT(rtb_out_n)), 5)))) + DINT_TO_UDINT(DWORD_TO_DINT(SHL(DINT_TO_DWORD(BOOL_TO_DINT(rtb_FL_boHVC_AllCellBalanced)), 4)))) + DINT_TO_UDINT(DWORD_TO_DINT(SHL(DINT_TO_DWORD(BOOL_TO_DINT(rtb_out_l)), 3)))) + DINT_TO_UDINT(DWORD_TO_DINT(SHL(DINT_TO_DWORD(BOOL_TO_DINT(rtb_IT_boUDC_KL15_C)), 2)))) + DINT_TO_UDINT(DWORD_TO_DINT(SHL(DINT_TO_DWORD(BOOL_TO_DINT(rtb_IT_boUDC_KL15_D)), 1)))) + BOOL_TO_UDINT(rtb_IT_boBMS_SDError_BB1));
        OP_ChiefMaster_IP_Msg1[1] := UDINT_TO_USINT(((((((DINT_TO_UDINT(DWORD_TO_DINT(SHL(DINT_TO_DWORD(BOOL_TO_DINT(rtb_IT_boHW_DCHV_Minus_FB)), 7))) + DINT_TO_UDINT(DWORD_TO_DINT(SHL(DINT_TO_DWORD(BOOL_TO_DINT(rtb_IT_boHW_DCHV_Plus_FB)), 6)))) + DINT_TO_UDINT(DWORD_TO_DINT(SHL(DINT_TO_DWORD(BOOL_TO_DINT(rtb_out_ne)), 5)))) + DINT_TO_UDINT(DWORD_TO_DINT(SHL(DINT_TO_DWORD(BOOL_TO_DINT(rtb_out_i)), 4)))) + DINT_TO_UDINT(DWORD_TO_DINT(SHL(DINT_TO_DWORD(BOOL_TO_DINT(rtb_IT_boHW_HVIL_BDU)), 3)))) + DINT_TO_UDINT(DWORD_TO_DINT(SHL(DINT_TO_DWORD(BOOL_TO_DINT(DI_ResetButton_LED_NO)), 2)))) + DINT_TO_UDINT(DWORD_TO_DINT(SHL(DINT_TO_DWORD(BOOL_TO_DINT(rtb_IT_boHW_EmergencyButton_NO)), 1)))) + BOOL_TO_UDINT(rtb_IT_sHW_EmergencyButton_NC));
        OP_ChiefMaster_IP_Msg1[3] := UINT_TO_USINT(DINT_TO_UINT(TRUNC(y_1)));
        OP_ChiefMaster_IP_Msg1[4] := DINT_TO_USINT(DWORD_TO_DINT(SHR(DINT_TO_DWORD(UINT_TO_DINT(DINT_TO_UINT(TRUNC(y_1)))), 8)));
        (* End of Outputs for SubSystem: '<Root>/ChiefMaster' *)
        OP_ChiefMaster_IP_Msg1[5] := 0;
        OP_ChiefMaster_IP_Msg1[6] := 0;
        OP_ChiefMaster_IP_Msg1[7] := 0;
        (* Outputs for Atomic SubSystem: '<Root>/ChiefMaster' *)
        (* Outport: '<Root>/OP_ChiefMaster_OP_Msg2' incorporates:
         *  ArithShift: '<S983>/Shift Arithmetic'
         *  ArithShift: '<S983>/Shift Arithmetic1'
         *  ArithShift: '<S983>/Shift Arithmetic2'
         *  ArithShift: '<S983>/Shift Arithmetic3'
         *  ArithShift: '<S983>/Shift Arithmetic4'
         *  ArithShift: '<S983>/Shift Arithmetic5'
         *  ArithShift: '<S983>/Shift Arithmetic6'
         *  Constant: '<S814>/Constant2'
         *  DataTypeConversion: '<S983>/Data Type Conversion'
         *  DataTypeConversion: '<S983>/Data Type Conversion1'
         *  DataTypeConversion: '<S983>/Data Type Conversion2'
         *  DataTypeConversion: '<S983>/Data Type Conversion3'
         *  DataTypeConversion: '<S983>/Data Type Conversion4'
         *  DataTypeConversion: '<S983>/Data Type Conversion5'
         *  DataTypeConversion: '<S983>/Data Type Conversion6'
         *  DataTypeConversion: '<S983>/Data Type Conversion7'
         *  Outport: '<Root>/DO_KL15_BB1'
         *  Outport: '<Root>/DO_KL15_BB2'
         *  Outport: '<Root>/DO_KL15_BB3'
         *  Sum: '<S983>/Add' *)
        OP_ChiefMaster_OP_Msg2[0] := UDINT_TO_USINT(((((((DINT_TO_UDINT(DWORD_TO_DINT(SHL(DINT_TO_DWORD(BOOL_TO_DINT(DO_boKL15_IMD_BB2)), 7))) + DINT_TO_UDINT(DWORD_TO_DINT(SHL(DINT_TO_DWORD(BOOL_TO_DINT(DO_boKL15_IMD_BB1)), 6)))) + DINT_TO_UDINT(DWORD_TO_DINT(SHL(DINT_TO_DWORD(BOOL_TO_DINT(DO_REQ_MainHV_ON_Precharge)), 5)))) + DINT_TO_UDINT(DWORD_TO_DINT(SHL(DINT_TO_DWORD(BOOL_TO_DINT(DO_REQ_MainHV_ON_PLUS)), 4)))) + DINT_TO_UDINT(DWORD_TO_DINT(SHL(DINT_TO_DWORD(BOOL_TO_DINT(DO_REQ_MainHV_ON_MINUS)), 3)))) + DINT_TO_UDINT(DWORD_TO_DINT(SHL(DINT_TO_DWORD(BOOL_TO_DINT(DO_KL15_BB3)), 2)))) + DINT_TO_UDINT(DWORD_TO_DINT(SHL(DINT_TO_DWORD(BOOL_TO_DINT(DO_KL15_BB2)), 1)))) + BOOL_TO_UDINT(DO_KL15_BB1));
        (* End of Outputs for SubSystem: '<Root>/ChiefMaster' *)
        OP_ChiefMaster_OP_Msg2[3] := 0;
        OP_ChiefMaster_OP_Msg2[4] := 0;
        OP_ChiefMaster_OP_Msg2[5] := 0;
        OP_ChiefMaster_OP_Msg2[6] := 0;
        OP_ChiefMaster_OP_Msg2[7] := 0;
        (* Outputs for Atomic SubSystem: '<Root>/ChiefMaster' *)
        (* Outputs for Atomic SubSystem: '<S676>/BatteryPackSignals' *)
        (* Outport: '<Root>/OP_ChiefMaster_SS1_Msg3' incorporates:
         *  ArithShift: '<S990>/Shift Arithmetic'
         *  ArithShift: '<S990>/Shift Arithmetic1'
         *  ArithShift: '<S990>/Shift Arithmetic2'
         *  ArithShift: '<S990>/Shift Arithmetic4'
         *  ArithShift: '<S990>/Shift Arithmetic5'
         *  ArithShift: '<S990>/Shift Arithmetic6'
         *  DataTypeConversion: '<S990>/Data Type Conversion'
         *  DataTypeConversion: '<S990>/Data Type Conversion1'
         *  DataTypeConversion: '<S990>/Data Type Conversion2'
         *  DataTypeConversion: '<S990>/Data Type Conversion5'
         *  DataTypeConversion: '<S990>/Data Type Conversion6'
         *  DataTypeConversion: '<S990>/Data Type Conversion7'
         *  Logic: '<S12>/OR'
         *  Logic: '<S12>/OR1'
         *  Logic: '<S12>/OR2'
         *  MinMax: '<S118>/Min'
         *  SignalConversion: '<S698>/Signal Copy'
         *  SignalConversion: '<S699>/Signal Copy'
         *  SignalConversion: '<S700>/Signal Copy'
         *  Sum: '<S117>/Add'
         *  Sum: '<S990>/Add' *)
        OP_ChiefMaster_SS1_Msg3[0] := UDINT_TO_USINT(((((((DINT_TO_UDINT(DWORD_TO_DINT(SHL(DINT_TO_DWORD(BOOL_TO_DINT(rtb_FL_boKL15_Disable)), 7))) + DINT_TO_UDINT(DWORD_TO_DINT(SHL(DINT_TO_DWORD(BOOL_TO_DINT(rtb_FL_boSS_BDU_Reset)), 6)))) + DINT_TO_UDINT(DWORD_TO_DINT(SHL(DINT_TO_DWORD(BOOL_TO_DINT(rtb_Delay_j)), 5)))) + USINT_TO_UDINT(rtb_ShiftArithmetic3_p)) + DINT_TO_UDINT(DWORD_TO_DINT(SHL(DINT_TO_DWORD(BOOL_TO_DINT(rtb_FL_boSS_System_Error)), 3)))) + DINT_TO_UDINT(DWORD_TO_DINT(SHL(DINT_TO_DWORD(BOOL_TO_DINT((rtb_IP_boBMS_SDError_BB1 OR rtb_IP_boBMS_SDError_BB2) OR rtb_IP_boBMS_SDError_BB3)), 2)))) + DINT_TO_UDINT(DWORD_TO_DINT(SHL(DINT_TO_DWORD(BOOL_TO_DINT((rtb_IT_boBMS_Error_BB1 OR rtb_IT_boBMS_Error_BB2) OR rtb_IT_boBMS_Error_BB3)), 1)))) + BOOL_TO_UDINT((rtb_IT_boBMS_Warning_BB1 OR rtb_IT_boBMS_Warning_BB2) OR rtb_IT_boBMS_Warning_BB3));
        (* End of Outputs for SubSystem: '<S676>/BatteryPackSignals' *)
        (* End of Outputs for SubSystem: '<Root>/ChiefMaster' *)
        OP_ChiefMaster_SS1_Msg3[3] := CMState_e2;
        (* Outputs for Atomic SubSystem: '<Root>/ChiefMaster' *)
        OP_ChiefMaster_SS1_Msg3[4] := UDINT_TO_USINT((BOOL_TO_UDINT(rtb_Switch_b) + BOOL_TO_UDINT(rtb_Switch1_fj)) + BOOL_TO_UDINT(rtb_Switch2_d));
        temp5 := MIN(rtb_ExtractDesiredBits_mi, rtb_ExtractDesiredBits_ebk);
        OP_ChiefMaster_SS1_Msg3[6] := MIN(temp5, rtb_ExtractDesiredBits_be);
        (* Outport: '<Root>/OP_ChiefMaster_SS2_Msg4' incorporates:
         *  DataTypeConversion: '<S1001>/Data Type Conversion2'
         *  DataTypeConversion: '<S1003>/Extract Desired Bits'
         *  DataTypeConversion: '<S1004>/Extract Desired Bits'
         *  DataTypeConversion: '<S1005>/Data Type Conversion2'
         *  DataTypeConversion: '<S1007>/Extract Desired Bits'
         *  DataTypeConversion: '<S1008>/Extract Desired Bits'
         *  DataTypeConversion: '<S1009>/Data Type Conversion2'
         *  DataTypeConversion: '<S1011>/Extract Desired Bits'
         *  DataTypeConversion: '<S1012>/Extract Desired Bits'
         *  DataTypeConversion: '<S1013>/Data Type Conversion2'
         *  DataTypeConversion: '<S1015>/Extract Desired Bits'
         *  DataTypeConversion: '<S1016>/Extract Desired Bits' *)
        OP_ChiefMaster_SS2_Msg4[0] := UINT_TO_USINT(DINT_TO_UINT(TRUNC(rtb_Add_nm)));
        OP_ChiefMaster_SS2_Msg4[1] := DINT_TO_USINT(DWORD_TO_DINT(SHR(DINT_TO_DWORD(UINT_TO_DINT(DINT_TO_UINT(TRUNC(rtb_Add_nm)))), 8)));
        OP_ChiefMaster_SS2_Msg4[2] := UINT_TO_USINT(DINT_TO_UINT(TRUNC(maxV)));
        OP_ChiefMaster_SS2_Msg4[3] := DINT_TO_USINT(DWORD_TO_DINT(SHR(DINT_TO_DWORD(UINT_TO_DINT(DINT_TO_UINT(TRUNC(maxV)))), 8)));
        OP_ChiefMaster_SS2_Msg4[4] := UINT_TO_USINT(DINT_TO_UINT(TRUNC(rtb_Add_d4)));
        OP_ChiefMaster_SS2_Msg4[5] := DINT_TO_USINT(DWORD_TO_DINT(SHR(DINT_TO_DWORD(UINT_TO_DINT(DINT_TO_UINT(TRUNC(rtb_Add_d4)))), 8)));
        OP_ChiefMaster_SS2_Msg4[6] := UINT_TO_USINT(DINT_TO_UINT(TRUNC(rtb_FL_sSS_MaxDisChargeCurrent)));
        OP_ChiefMaster_SS2_Msg4[7] := DINT_TO_USINT(DWORD_TO_DINT(SHR(DINT_TO_DWORD(UINT_TO_DINT(DINT_TO_UINT(TRUNC(rtb_FL_sSS_MaxDisChargeCurrent)))), 8)));
        (* Outport: '<Root>/OP_ChiefMaster_Calc_Msg5' incorporates:
         *  DataTypeConversion: '<S832>/Data Type Conversion2'
         *  DataTypeConversion: '<S834>/Extract Desired Bits'
         *  DataTypeConversion: '<S835>/Extract Desired Bits'
         *  DataTypeConversion: '<S836>/Data Type Conversion2'
         *  DataTypeConversion: '<S838>/Extract Desired Bits'
         *  DataTypeConversion: '<S839>/Extract Desired Bits'
         *  DataTypeConversion: '<S840>/Data Type Conversion2'
         *  DataTypeConversion: '<S842>/Extract Desired Bits'
         *  DataTypeConversion: '<S843>/Extract Desired Bits'
         *  DataTypeConversion: '<S844>/Data Type Conversion2'
         *  DataTypeConversion: '<S846>/Extract Desired Bits'
         *  DataTypeConversion: '<S847>/Extract Desired Bits' *)
        OP_ChiefMaster_Calc_Msg5[0] := UINT_TO_USINT(DINT_TO_UINT(TRUNC(rtb_Abs)));
        OP_ChiefMaster_Calc_Msg5[1] := DINT_TO_USINT(DWORD_TO_DINT(SHR(DINT_TO_DWORD(UINT_TO_DINT(DINT_TO_UINT(TRUNC(rtb_Abs)))), 8)));
        OP_ChiefMaster_Calc_Msg5[2] := UINT_TO_USINT(DINT_TO_UINT(TRUNC(rtb_Abs1)));
        OP_ChiefMaster_Calc_Msg5[3] := DINT_TO_USINT(DWORD_TO_DINT(SHR(DINT_TO_DWORD(UINT_TO_DINT(DINT_TO_UINT(TRUNC(rtb_Abs1)))), 8)));
        OP_ChiefMaster_Calc_Msg5[4] := UINT_TO_USINT(DINT_TO_UINT(TRUNC(rtb_Abs2)));
        OP_ChiefMaster_Calc_Msg5[5] := DINT_TO_USINT(DWORD_TO_DINT(SHR(DINT_TO_DWORD(UINT_TO_DINT(DINT_TO_UINT(TRUNC(rtb_Abs2)))), 8)));
        OP_ChiefMaster_Calc_Msg5[6] := UINT_TO_USINT(DINT_TO_UINT(TRUNC(rtb_UnitDelay)));
        OP_ChiefMaster_Calc_Msg5[7] := DINT_TO_USINT(DWORD_TO_DINT(SHR(DINT_TO_DWORD(UINT_TO_DINT(DINT_TO_UINT(TRUNC(rtb_UnitDelay)))), 8)));
        (* Outport: '<Root>/OP_ChiefMaster_BDU_Msg6' incorporates:
         *  Constant: '<S803>/Constant1'
         *  DataTypeConversion: '<S848>/Data Type Conversion2'
         *  DataTypeConversion: '<S850>/Extract Desired Bits'
         *  DataTypeConversion: '<S851>/Extract Desired Bits'
         *  DataTypeConversion: '<S852>/Data Type Conversion2'
         *  DataTypeConversion: '<S854>/Extract Desired Bits'
         *  DataTypeConversion: '<S855>/Extract Desired Bits' *)
        OP_ChiefMaster_BDU_Msg6[0] := UINT_TO_USINT(DINT_TO_UINT(TRUNC(rtb_Divide1_p)));
        OP_ChiefMaster_BDU_Msg6[1] := DINT_TO_USINT(DWORD_TO_DINT(SHR(DINT_TO_DWORD(UINT_TO_DINT(DINT_TO_UINT(TRUNC(rtb_Divide1_p)))), 8)));
        OP_ChiefMaster_BDU_Msg6[2] := UINT_TO_USINT(DINT_TO_UINT(TRUNC(rtb_Divide2)));
        OP_ChiefMaster_BDU_Msg6[3] := DINT_TO_USINT(DWORD_TO_DINT(SHR(DINT_TO_DWORD(UINT_TO_DINT(DINT_TO_UINT(TRUNC(rtb_Divide2)))), 8)));
        (* End of Outputs for SubSystem: '<Root>/ChiefMaster' *)
        OP_ChiefMaster_BDU_Msg6[7] := 0;
        (* Outputs for Atomic SubSystem: '<Root>/ChiefMaster' *)
        (* Outputs for Atomic SubSystem: '<S676>/BatteryPackSignals' *)
        (* Outport: '<Root>/OP_ChiefMaster_Battery1_Msg7' incorporates:
         *  ArithShift: '<S861>/Shift Arithmetic'
         *  ArithShift: '<S861>/Shift Arithmetic1'
         *  ArithShift: '<S861>/Shift Arithmetic2'
         *  ArithShift: '<S861>/Shift Arithmetic3'
         *  ArithShift: '<S861>/Shift Arithmetic4'
         *  ArithShift: '<S861>/Shift Arithmetic5'
         *  ArithShift: '<S861>/Shift Arithmetic6'
         *  DataTypeConversion: '<S804>/Data Type Conversion1'
         *  DataTypeConversion: '<S858>/Data Type Conversion2'
         *  DataTypeConversion: '<S859>/Data Type Conversion2'
         *  DataTypeConversion: '<S861>/Data Type Conversion'
         *  DataTypeConversion: '<S861>/Data Type Conversion1'
         *  DataTypeConversion: '<S861>/Data Type Conversion2'
         *  DataTypeConversion: '<S861>/Data Type Conversion4'
         *  DataTypeConversion: '<S861>/Data Type Conversion5'
         *  DataTypeConversion: '<S861>/Data Type Conversion6'
         *  DataTypeConversion: '<S861>/Data Type Conversion7'
         *  DataTypeConversion: '<S864>/Extract Desired Bits'
         *  DataTypeConversion: '<S865>/Extract Desired Bits'
         *  DataTypeConversion: '<S866>/Extract Desired Bits'
         *  DataTypeConversion: '<S867>/Extract Desired Bits'
         *  SignalConversion: '<S682>/BusConversion_InsertedFor_IT_BatterySignal_Databus_at_inport_0'
         *  Sum: '<S861>/Add' *)
        OP_ChiefMaster_Battery1_Msg7[1] := UDINT_TO_USINT(((((((DINT_TO_UDINT(DWORD_TO_DINT(SHL(DINT_TO_DWORD(BOOL_TO_DINT(rtb_IT_boBMS_Warning_BB1)), 7))) + DINT_TO_UDINT(DWORD_TO_DINT(SHL(DINT_TO_DWORD(BOOL_TO_DINT(rtb_IT_boBMS_Error_BB1)), 6)))) + DINT_TO_UDINT(DWORD_TO_DINT(SHL(DINT_TO_DWORD(BOOL_TO_DINT(rtb_IP_boBMS_IMD_Active_BB1)), 5)))) + DINT_TO_UDINT(DWORD_TO_DINT(SHL(DINT_TO_DWORD(BOOL_TO_DINT(rtb_AND_l2)), 4)))) + DINT_TO_UDINT(DWORD_TO_DINT(SHL(DINT_TO_DWORD(BOOL_TO_DINT(rtb_S_in)), 3)))) + DINT_TO_UDINT(DWORD_TO_DINT(SHL(DINT_TO_DWORD(BOOL_TO_DINT(rtb_IP_boBMS_HV_Plus_Sense_BB1)), 2)))) + DINT_TO_UDINT(DWORD_TO_DINT(SHL(DINT_TO_DWORD(BOOL_TO_DINT(rtb_IP_boBMS_HV_Minus_Sense_BB1)), 1)))) + BOOL_TO_UDINT(rtb_IP_boBMS_HV_REL_ON_BB1));
        (* End of Outputs for SubSystem: '<S676>/BatteryPackSignals' *)
        OP_ChiefMaster_Battery1_Msg7[2] := UINT_TO_USINT(DINT_TO_UINT(TRUNC(rtb_Switch3)));
        OP_ChiefMaster_Battery1_Msg7[3] := DINT_TO_USINT(DWORD_TO_DINT(SHR(DINT_TO_DWORD(UINT_TO_DINT(DINT_TO_UINT(TRUNC(rtb_Switch3)))), 8)));
        OP_ChiefMaster_Battery1_Msg7[4] := UINT_TO_USINT(DINT_TO_UINT(TRUNC(rtb_Switch_a)));
        OP_ChiefMaster_Battery1_Msg7[5] := DINT_TO_USINT(DWORD_TO_DINT(SHR(DINT_TO_DWORD(UINT_TO_DINT(DINT_TO_UINT(TRUNC(rtb_Switch_a)))), 8)));
        (* Outputs for Atomic SubSystem: '<S676>/BatteryPackSignals' *)
        OP_ChiefMaster_Battery1_Msg7[6] := rtb_DataTypeConversion_k;
        (* End of Outputs for SubSystem: '<S676>/BatteryPackSignals' *)
        OP_ChiefMaster_Battery1_Msg7[7] := DINT_TO_USINT(TRUNC(rtb_IT_sBMS_InternalResistance_BB1_ohms));
        (* Outport: '<Root>/OP_ChiefMaster_Battery1_Msg8' incorporates:
         *  DataTypeConversion: '<S868>/Data Type Conversion2'
         *  DataTypeConversion: '<S869>/Data Type Conversion2'
         *  DataTypeConversion: '<S870>/Data Type Conversion2'
         *  DataTypeConversion: '<S871>/Data Type Conversion2'
         *  DataTypeConversion: '<S876>/Extract Desired Bits'
         *  DataTypeConversion: '<S877>/Extract Desired Bits'
         *  DataTypeConversion: '<S878>/Extract Desired Bits'
         *  DataTypeConversion: '<S879>/Extract Desired Bits'
         *  DataTypeConversion: '<S880>/Extract Desired Bits'
         *  DataTypeConversion: '<S881>/Extract Desired Bits'
         *  DataTypeConversion: '<S882>/Extract Desired Bits'
         *  DataTypeConversion: '<S883>/Extract Desired Bits' *)
        OP_ChiefMaster_Battery1_Msg8[0] := UINT_TO_USINT(DINT_TO_UINT(TRUNC(rtb_Add_b)));
        OP_ChiefMaster_Battery1_Msg8[1] := DINT_TO_USINT(DWORD_TO_DINT(SHR(DINT_TO_DWORD(UINT_TO_DINT(DINT_TO_UINT(TRUNC(rtb_Add_b)))), 8)));
        OP_ChiefMaster_Battery1_Msg8[2] := UINT_TO_USINT(DINT_TO_UINT(TRUNC(rtb_Add_ic5)));
        OP_ChiefMaster_Battery1_Msg8[3] := DINT_TO_USINT(DWORD_TO_DINT(SHR(DINT_TO_DWORD(UINT_TO_DINT(DINT_TO_UINT(TRUNC(rtb_Add_ic5)))), 8)));
        OP_ChiefMaster_Battery1_Msg8[4] := UINT_TO_USINT(DINT_TO_UINT(TRUNC(rtb_Min)));
        OP_ChiefMaster_Battery1_Msg8[5] := DINT_TO_USINT(DWORD_TO_DINT(SHR(DINT_TO_DWORD(UINT_TO_DINT(DINT_TO_UINT(TRUNC(rtb_Min)))), 8)));
        OP_ChiefMaster_Battery1_Msg8[6] := UINT_TO_USINT(DINT_TO_UINT(TRUNC(rtb_Add_psl)));
        OP_ChiefMaster_Battery1_Msg8[7] := DINT_TO_USINT(DWORD_TO_DINT(SHR(DINT_TO_DWORD(UINT_TO_DINT(DINT_TO_UINT(TRUNC(rtb_Add_psl)))), 8)));
        (* Outputs for Atomic SubSystem: '<S676>/BatteryPackSignals' *)
        (* Outport: '<Root>/OP_ChiefMaster_Battery1_Msg9' incorporates:
         *  Constant: '<S806>/Constant1'
         *  Constant: '<S806>/Constant2'
         *  Constant: '<S806>/Constant9'
         *  DataTypeConversion: '<S806>/Data Type Conversion'
         *  DataTypeConversion: '<S806>/Data Type Conversion1'
         *  DataTypeConversion: '<S884>/Data Type Conversion2'
         *  DataTypeConversion: '<S885>/Data Type Conversion2'
         *  DataTypeConversion: '<S890>/Extract Desired Bits'
         *  DataTypeConversion: '<S891>/Extract Desired Bits'
         *  DataTypeConversion: '<S892>/Extract Desired Bits'
         *  DataTypeConversion: '<S893>/Extract Desired Bits'
         *  SignalConversion: '<S682>/BusConversion_InsertedFor_IT_BatterySignal_Databus_at_inport_0'
         *  Sum: '<S886>/Add'
         *  Sum: '<S887>/Add' *)
        OP_ChiefMaster_Battery1_Msg9[0] := DINT_TO_USINT(TRUNC(rtb_Add_no - -40.0));
        OP_ChiefMaster_Battery1_Msg9[1] := DINT_TO_USINT(TRUNC(rtb_Add_a5 - -40.0));
        (* End of Outputs for SubSystem: '<S676>/BatteryPackSignals' *)
        OP_ChiefMaster_Battery1_Msg9[2] := UINT_TO_USINT(DINT_TO_UINT(TRUNC(rtb_Switch2_k)));
        OP_ChiefMaster_Battery1_Msg9[3] := DINT_TO_USINT(DWORD_TO_DINT(SHR(DINT_TO_DWORD(UINT_TO_DINT(DINT_TO_UINT(TRUNC(rtb_Switch2_k)))), 8)));
        OP_ChiefMaster_Battery1_Msg9[4] := UINT_TO_USINT(DINT_TO_UINT(TRUNC(rtb_Add_ie)));
        OP_ChiefMaster_Battery1_Msg9[5] := DINT_TO_USINT(DWORD_TO_DINT(SHR(DINT_TO_DWORD(UINT_TO_DINT(DINT_TO_UINT(TRUNC(rtb_Add_ie)))), 8)));
        (* End of Outputs for SubSystem: '<Root>/ChiefMaster' *)
        OP_ChiefMaster_Battery1_Msg9[6] := 0;
        OP_ChiefMaster_Battery1_Msg9[7] := 0;
        (* Outputs for Atomic SubSystem: '<Root>/ChiefMaster' *)
        (* Outputs for Atomic SubSystem: '<S676>/BatteryPackSignals' *)
        (* Outport: '<Root>/OP_ChiefMaster_Battery2_Msg10' incorporates:
         *  ArithShift: '<S899>/Shift Arithmetic'
         *  ArithShift: '<S899>/Shift Arithmetic1'
         *  ArithShift: '<S899>/Shift Arithmetic2'
         *  ArithShift: '<S899>/Shift Arithmetic3'
         *  ArithShift: '<S899>/Shift Arithmetic4'
         *  ArithShift: '<S899>/Shift Arithmetic5'
         *  ArithShift: '<S899>/Shift Arithmetic6'
         *  DataTypeConversion: '<S807>/Data Type Conversion'
         *  DataTypeConversion: '<S896>/Data Type Conversion2'
         *  DataTypeConversion: '<S897>/Data Type Conversion2'
         *  DataTypeConversion: '<S899>/Data Type Conversion'
         *  DataTypeConversion: '<S899>/Data Type Conversion1'
         *  DataTypeConversion: '<S899>/Data Type Conversion2'
         *  DataTypeConversion: '<S899>/Data Type Conversion4'
         *  DataTypeConversion: '<S899>/Data Type Conversion5'
         *  DataTypeConversion: '<S899>/Data Type Conversion6'
         *  DataTypeConversion: '<S899>/Data Type Conversion7'
         *  DataTypeConversion: '<S902>/Extract Desired Bits'
         *  DataTypeConversion: '<S903>/Extract Desired Bits'
         *  DataTypeConversion: '<S904>/Extract Desired Bits'
         *  DataTypeConversion: '<S905>/Extract Desired Bits'
         *  SignalConversion: '<S682>/BusConversion_InsertedFor_IT_BatterySignal_Databus_at_inport_0'
         *  Sum: '<S899>/Add' *)
        OP_ChiefMaster_Battery2_Msg10[1] := UDINT_TO_USINT(((((((DINT_TO_UDINT(DWORD_TO_DINT(SHL(DINT_TO_DWORD(BOOL_TO_DINT(rtb_IT_boBMS_Warning_BB2)), 7))) + DINT_TO_UDINT(DWORD_TO_DINT(SHL(DINT_TO_DWORD(BOOL_TO_DINT(rtb_IT_boBMS_Error_BB2)), 6)))) + DINT_TO_UDINT(DWORD_TO_DINT(SHL(DINT_TO_DWORD(BOOL_TO_DINT(rtb_IP_boBMS_IMD_Active_BB2)), 5)))) + DINT_TO_UDINT(DWORD_TO_DINT(SHL(DINT_TO_DWORD(BOOL_TO_DINT(rtb_AND_ni)), 4)))) + DINT_TO_UDINT(DWORD_TO_DINT(SHL(DINT_TO_DWORD(BOOL_TO_DINT(rtb_IP_boBatt1_Actia_Availability)), 3)))) + DINT_TO_UDINT(DWORD_TO_DINT(SHL(DINT_TO_DWORD(BOOL_TO_DINT(rtb_IP_boBMS_HV_Plus_Sense_BB2)), 2)))) + DINT_TO_UDINT(DWORD_TO_DINT(SHL(DINT_TO_DWORD(BOOL_TO_DINT(rtb_IP_boBMS_HV_Minus_Sense_BB2)), 1)))) + BOOL_TO_UDINT(rtb_IP_boBMS_HV_REL_ON_BB2));
        (* End of Outputs for SubSystem: '<S676>/BatteryPackSignals' *)
        OP_ChiefMaster_Battery2_Msg10[2] := UINT_TO_USINT(DINT_TO_UINT(TRUNC(rtb_Add_an)));
        OP_ChiefMaster_Battery2_Msg10[3] := DINT_TO_USINT(DWORD_TO_DINT(SHR(DINT_TO_DWORD(UINT_TO_DINT(DINT_TO_UINT(TRUNC(rtb_Add_an)))), 8)));
        OP_ChiefMaster_Battery2_Msg10[4] := UINT_TO_USINT(DINT_TO_UINT(TRUNC(rtb_Add_ci)));
        OP_ChiefMaster_Battery2_Msg10[5] := DINT_TO_USINT(DWORD_TO_DINT(SHR(DINT_TO_DWORD(UINT_TO_DINT(DINT_TO_UINT(TRUNC(rtb_Add_ci)))), 8)));
        (* Outputs for Atomic SubSystem: '<S676>/BatteryPackSignals' *)
        OP_ChiefMaster_Battery2_Msg10[6] := rtb_DataTypeConversion1;
        (* End of Outputs for SubSystem: '<S676>/BatteryPackSignals' *)
        OP_ChiefMaster_Battery2_Msg10[7] := DINT_TO_USINT(TRUNC(rtb_Add_c0));
        (* Outport: '<Root>/OP_ChiefMaster_Battery2_Msg11' incorporates:
         *  DataTypeConversion: '<S906>/Data Type Conversion2'
         *  DataTypeConversion: '<S907>/Data Type Conversion2'
         *  DataTypeConversion: '<S908>/Data Type Conversion2'
         *  DataTypeConversion: '<S909>/Data Type Conversion2'
         *  DataTypeConversion: '<S914>/Extract Desired Bits'
         *  DataTypeConversion: '<S915>/Extract Desired Bits'
         *  DataTypeConversion: '<S916>/Extract Desired Bits'
         *  DataTypeConversion: '<S917>/Extract Desired Bits'
         *  DataTypeConversion: '<S918>/Extract Desired Bits'
         *  DataTypeConversion: '<S919>/Extract Desired Bits'
         *  DataTypeConversion: '<S920>/Extract Desired Bits'
         *  DataTypeConversion: '<S921>/Extract Desired Bits' *)
        OP_ChiefMaster_Battery2_Msg11[0] := UINT_TO_USINT(DINT_TO_UINT(TRUNC(rtb_Add_h)));
        OP_ChiefMaster_Battery2_Msg11[1] := DINT_TO_USINT(DWORD_TO_DINT(SHR(DINT_TO_DWORD(UINT_TO_DINT(DINT_TO_UINT(TRUNC(rtb_Add_h)))), 8)));
        OP_ChiefMaster_Battery2_Msg11[2] := UINT_TO_USINT(DINT_TO_UINT(TRUNC(rtb_Add_kf)));
        OP_ChiefMaster_Battery2_Msg11[3] := DINT_TO_USINT(DWORD_TO_DINT(SHR(DINT_TO_DWORD(UINT_TO_DINT(DINT_TO_UINT(TRUNC(rtb_Add_kf)))), 8)));
        OP_ChiefMaster_Battery2_Msg11[4] := UINT_TO_USINT(DINT_TO_UINT(TRUNC(rtb_Add_cv)));
        OP_ChiefMaster_Battery2_Msg11[5] := DINT_TO_USINT(DWORD_TO_DINT(SHR(DINT_TO_DWORD(UINT_TO_DINT(DINT_TO_UINT(TRUNC(rtb_Add_cv)))), 8)));
        OP_ChiefMaster_Battery2_Msg11[6] := UINT_TO_USINT(DINT_TO_UINT(TRUNC(rtb_Add_ic)));
        OP_ChiefMaster_Battery2_Msg11[7] := DINT_TO_USINT(DWORD_TO_DINT(SHR(DINT_TO_DWORD(UINT_TO_DINT(DINT_TO_UINT(TRUNC(rtb_Add_ic)))), 8)));
        (* Outputs for Atomic SubSystem: '<S676>/BatteryPackSignals' *)
        (* Outport: '<Root>/OP_ChiefMaster_Battery2_Msg12' incorporates:
         *  Constant: '<S809>/Constant1'
         *  Constant: '<S809>/Constant2'
         *  Constant: '<S809>/Constant9'
         *  DataTypeConversion: '<S809>/Data Type Conversion'
         *  DataTypeConversion: '<S809>/Data Type Conversion1'
         *  DataTypeConversion: '<S922>/Data Type Conversion2'
         *  DataTypeConversion: '<S923>/Data Type Conversion2'
         *  DataTypeConversion: '<S928>/Extract Desired Bits'
         *  DataTypeConversion: '<S929>/Extract Desired Bits'
         *  DataTypeConversion: '<S930>/Extract Desired Bits'
         *  DataTypeConversion: '<S931>/Extract Desired Bits'
         *  SignalConversion: '<S682>/BusConversion_InsertedFor_IT_BatterySignal_Databus_at_inport_0'
         *  Sum: '<S924>/Add'
         *  Sum: '<S925>/Add' *)
        OP_ChiefMaster_Battery2_Msg12[0] := DINT_TO_USINT(TRUNC(rtb_Add_g4 - -40.0));
        OP_ChiefMaster_Battery2_Msg12[1] := DINT_TO_USINT(TRUNC(rtb_Add_i5o - -40.0));
        (* End of Outputs for SubSystem: '<S676>/BatteryPackSignals' *)
        OP_ChiefMaster_Battery2_Msg12[2] := UINT_TO_USINT(DINT_TO_UINT(TRUNC(rtb_Divide_i)));
        OP_ChiefMaster_Battery2_Msg12[3] := DINT_TO_USINT(DWORD_TO_DINT(SHR(DINT_TO_DWORD(UINT_TO_DINT(DINT_TO_UINT(TRUNC(rtb_Divide_i)))), 8)));
        OP_ChiefMaster_Battery2_Msg12[4] := UINT_TO_USINT(DINT_TO_UINT(TRUNC(rtb_Add_oy)));
        OP_ChiefMaster_Battery2_Msg12[5] := DINT_TO_USINT(DWORD_TO_DINT(SHR(DINT_TO_DWORD(UINT_TO_DINT(DINT_TO_UINT(TRUNC(rtb_Add_oy)))), 8)));
        (* End of Outputs for SubSystem: '<Root>/ChiefMaster' *)
        OP_ChiefMaster_Battery2_Msg12[6] := 0;
        OP_ChiefMaster_Battery2_Msg12[7] := 0;
        (* Outputs for Atomic SubSystem: '<Root>/ChiefMaster' *)
        (* Outputs for Atomic SubSystem: '<S676>/BatteryPackSignals' *)
        (* Outport: '<Root>/OP_ChiefMaster_Battery3_Msg13' incorporates:
         *  ArithShift: '<S936>/Shift Arithmetic'
         *  ArithShift: '<S936>/Shift Arithmetic1'
         *  ArithShift: '<S936>/Shift Arithmetic2'
         *  ArithShift: '<S936>/Shift Arithmetic3'
         *  ArithShift: '<S936>/Shift Arithmetic4'
         *  ArithShift: '<S936>/Shift Arithmetic5'
         *  ArithShift: '<S936>/Shift Arithmetic6'
         *  DataTypeConversion: '<S810>/Data Type Conversion1'
         *  DataTypeConversion: '<S934>/Data Type Conversion2'
         *  DataTypeConversion: '<S935>/Data Type Conversion2'
         *  DataTypeConversion: '<S936>/Data Type Conversion'
         *  DataTypeConversion: '<S936>/Data Type Conversion1'
         *  DataTypeConversion: '<S936>/Data Type Conversion2'
         *  DataTypeConversion: '<S936>/Data Type Conversion4'
         *  DataTypeConversion: '<S936>/Data Type Conversion5'
         *  DataTypeConversion: '<S936>/Data Type Conversion6'
         *  DataTypeConversion: '<S936>/Data Type Conversion7'
         *  DataTypeConversion: '<S940>/Extract Desired Bits'
         *  DataTypeConversion: '<S941>/Extract Desired Bits'
         *  DataTypeConversion: '<S942>/Extract Desired Bits'
         *  DataTypeConversion: '<S943>/Extract Desired Bits'
         *  SignalConversion: '<S682>/BusConversion_InsertedFor_IT_BatterySignal_Databus_at_inport_0'
         *  Sum: '<S936>/Add' *)
        OP_ChiefMaster_Battery3_Msg13[1] := UDINT_TO_USINT(((((((DINT_TO_UDINT(DWORD_TO_DINT(SHL(DINT_TO_DWORD(BOOL_TO_DINT(rtb_IT_boBMS_Warning_BB3)), 7))) + DINT_TO_UDINT(DWORD_TO_DINT(SHL(DINT_TO_DWORD(BOOL_TO_DINT(rtb_IT_boBMS_Error_BB3)), 6)))) + DINT_TO_UDINT(DWORD_TO_DINT(SHL(DINT_TO_DWORD(BOOL_TO_DINT(rtb_IP_boBMS_IMD_Active_BB3)), 5)))) + DINT_TO_UDINT(DWORD_TO_DINT(SHL(DINT_TO_DWORD(BOOL_TO_DINT(rtb_AND_ma)), 4)))) + DINT_TO_UDINT(DWORD_TO_DINT(SHL(DINT_TO_DWORD(BOOL_TO_DINT(rtb_Delay_dl)), 3)))) + DINT_TO_UDINT(DWORD_TO_DINT(SHL(DINT_TO_DWORD(BOOL_TO_DINT(rtb_IP_boBMS_HV_Plus_Sense_BB3)), 2)))) + DINT_TO_UDINT(DWORD_TO_DINT(SHL(DINT_TO_DWORD(BOOL_TO_DINT(rtb_IP_boBMS_HV_Minus_Sense_BB3)), 1)))) + BOOL_TO_UDINT(rtb_IP_boBMS_HV_REL_ON_BB3));
        (* End of Outputs for SubSystem: '<S676>/BatteryPackSignals' *)
        OP_ChiefMaster_Battery3_Msg13[2] := UINT_TO_USINT(DINT_TO_UINT(TRUNC(rtb_Add_e)));
        OP_ChiefMaster_Battery3_Msg13[3] := DINT_TO_USINT(DWORD_TO_DINT(SHR(DINT_TO_DWORD(UINT_TO_DINT(DINT_TO_UINT(TRUNC(rtb_Add_e)))), 8)));
        OP_ChiefMaster_Battery3_Msg13[4] := UINT_TO_USINT(DINT_TO_UINT(TRUNC(rtb_Switch5_bs)));
        OP_ChiefMaster_Battery3_Msg13[5] := DINT_TO_USINT(DWORD_TO_DINT(SHR(DINT_TO_DWORD(UINT_TO_DINT(DINT_TO_UINT(TRUNC(rtb_Switch5_bs)))), 8)));
        (* Outputs for Atomic SubSystem: '<S676>/BatteryPackSignals' *)
        OP_ChiefMaster_Battery3_Msg13[6] := rtb_DataTypeConversion2_h;
        (* End of Outputs for SubSystem: '<S676>/BatteryPackSignals' *)
        OP_ChiefMaster_Battery3_Msg13[7] := DINT_TO_USINT(TRUNC(rtb_Add_egs));
        (* Outport: '<Root>/OP_ChiefMaster_Battery3_Msg14' incorporates:
         *  DataTypeConversion: '<S944>/Data Type Conversion2'
         *  DataTypeConversion: '<S945>/Data Type Conversion2'
         *  DataTypeConversion: '<S946>/Data Type Conversion2'
         *  DataTypeConversion: '<S947>/Data Type Conversion2'
         *  DataTypeConversion: '<S952>/Extract Desired Bits'
         *  DataTypeConversion: '<S953>/Extract Desired Bits'
         *  DataTypeConversion: '<S954>/Extract Desired Bits'
         *  DataTypeConversion: '<S955>/Extract Desired Bits'
         *  DataTypeConversion: '<S956>/Extract Desired Bits'
         *  DataTypeConversion: '<S957>/Extract Desired Bits'
         *  DataTypeConversion: '<S958>/Extract Desired Bits'
         *  DataTypeConversion: '<S959>/Extract Desired Bits' *)
        OP_ChiefMaster_Battery3_Msg14[0] := UINT_TO_USINT(DINT_TO_UINT(TRUNC(rtb_Add_g)));
        OP_ChiefMaster_Battery3_Msg14[1] := DINT_TO_USINT(DWORD_TO_DINT(SHR(DINT_TO_DWORD(UINT_TO_DINT(DINT_TO_UINT(TRUNC(rtb_Add_g)))), 8)));
        OP_ChiefMaster_Battery3_Msg14[2] := UINT_TO_USINT(DINT_TO_UINT(TRUNC(rtb_Add_j3)));
        OP_ChiefMaster_Battery3_Msg14[3] := DINT_TO_USINT(DWORD_TO_DINT(SHR(DINT_TO_DWORD(UINT_TO_DINT(DINT_TO_UINT(TRUNC(rtb_Add_j3)))), 8)));
        OP_ChiefMaster_Battery3_Msg14[4] := UINT_TO_USINT(DINT_TO_UINT(TRUNC(rtb_Add_d)));
        OP_ChiefMaster_Battery3_Msg14[5] := DINT_TO_USINT(DWORD_TO_DINT(SHR(DINT_TO_DWORD(UINT_TO_DINT(DINT_TO_UINT(TRUNC(rtb_Add_d)))), 8)));
        OP_ChiefMaster_Battery3_Msg14[6] := UINT_TO_USINT(DINT_TO_UINT(TRUNC(rtb_Add_en)));
        OP_ChiefMaster_Battery3_Msg14[7] := DINT_TO_USINT(DWORD_TO_DINT(SHR(DINT_TO_DWORD(UINT_TO_DINT(DINT_TO_UINT(TRUNC(rtb_Add_en)))), 8)));
        (* Outputs for Atomic SubSystem: '<S676>/BatteryPackSignals' *)
        (* Outport: '<Root>/OP_ChiefMaster_Battery3_Msg15' incorporates:
         *  Constant: '<S812>/Constant1'
         *  Constant: '<S812>/Constant2'
         *  Constant: '<S812>/Constant9'
         *  DataTypeConversion: '<S812>/Data Type Conversion'
         *  DataTypeConversion: '<S812>/Data Type Conversion1'
         *  DataTypeConversion: '<S960>/Data Type Conversion2'
         *  DataTypeConversion: '<S961>/Data Type Conversion2'
         *  DataTypeConversion: '<S966>/Extract Desired Bits'
         *  DataTypeConversion: '<S967>/Extract Desired Bits'
         *  DataTypeConversion: '<S968>/Extract Desired Bits'
         *  DataTypeConversion: '<S969>/Extract Desired Bits'
         *  SignalConversion: '<S682>/BusConversion_InsertedFor_IT_BatterySignal_Databus_at_inport_0'
         *  Sum: '<S962>/Add'
         *  Sum: '<S963>/Add' *)
        OP_ChiefMaster_Battery3_Msg15[0] := DINT_TO_USINT(TRUNC(rtb_Add_pi - -40.0));
        OP_ChiefMaster_Battery3_Msg15[1] := DINT_TO_USINT(TRUNC(rtb_Add_eo - -40.0));
        (* End of Outputs for SubSystem: '<S676>/BatteryPackSignals' *)
        OP_ChiefMaster_Battery3_Msg15[2] := UINT_TO_USINT(DINT_TO_UINT(TRUNC(rtb_Add_ky)));
        OP_ChiefMaster_Battery3_Msg15[3] := DINT_TO_USINT(DWORD_TO_DINT(SHR(DINT_TO_DWORD(UINT_TO_DINT(DINT_TO_UINT(TRUNC(rtb_Add_ky)))), 8)));
        OP_ChiefMaster_Battery3_Msg15[4] := UINT_TO_USINT(DINT_TO_UINT(TRUNC(rtb_Add_bh)));
        OP_ChiefMaster_Battery3_Msg15[5] := DINT_TO_USINT(DWORD_TO_DINT(SHR(DINT_TO_DWORD(UINT_TO_DINT(DINT_TO_UINT(TRUNC(rtb_Add_bh)))), 8)));
        (* End of Outputs for SubSystem: '<Root>/ChiefMaster' *)
        OP_ChiefMaster_Battery3_Msg15[6] := 0;
        OP_ChiefMaster_Battery3_Msg15[7] := 0;
END_CASE;

END_FUNCTION_BLOCK

// Device/Application/Chart
FUNCTION_BLOCK Chart
VAR_INPUT
	ssMethodType: SINT;
	In: BOOL;
END_VAR
VAR_OUTPUT
	Out: BOOL;
END_VAR
VAR
	is_c3_ChiefMaster: USINT;
	temporalCounter_i1: PLC_CODER_TIMER;
	is_active_c3_ChiefMaster: USINT;
END_VAR



CASE ssMethodType OF
    SS_INITIALIZE: 
        temporalCounter_i1(timerAction := 1, maxTime := 0);
        is_active_c3_ChiefMaster := 0;
        is_c3_ChiefMaster := ChiefMaster_IN_NO_ACTIVE_CHILD_j;
        Out := FALSE;
    SS_OUTPUT: 
        (* Chart: '<S48>/Chart' *)
        (* Gateway: ChiefMaster/Flow Logic/IMD Control/InsulationMonitoringReq/Chart *)
        (* During: ChiefMaster/Flow Logic/IMD Control/InsulationMonitoringReq/Chart *)

        IF is_active_c3_ChiefMaster = 0 THEN 
            (* Entry: ChiefMaster/Flow Logic/IMD Control/InsulationMonitoringReq/Chart *)
            is_active_c3_ChiefMaster := 1;
            (* Entry Internal: ChiefMaster/Flow Logic/IMD Control/InsulationMonitoringReq/Chart *)
            (* Transition: '<S49>:2' *)
            is_c3_ChiefMaster := ChiefMaster_IN_Default_e;
            (* Entry 'Default': '<S49>:1' *)
            (* '<S49>:1:2' Out = false *)
            Out := FALSE;
        ELSE 

            CASE is_c3_ChiefMaster OF
                ChiefMaster_IN_Actual: 
                    (* During 'Actual': '<S49>:7' *)
                    (* '<S49>:10:1' sf_internal_predicateOutput = In==false; *)

                    IF  NOT In THEN 
                        (* Transition: '<S49>:10' *)
                        is_c3_ChiefMaster := ChiefMaster_IN_Default_e;
                        (* Entry 'Default': '<S49>:1' *)
                        (* '<S49>:1:2' Out = false *)
                        Out := FALSE;
                    ELSE 
                        (* '<S49>:7:2' Out = In *)
                        Out := TRUE;
                    END_IF;

                ChiefMaster_IN_Default_e: 
                    (* During 'Default': '<S49>:1' *)
                    (* '<S49>:5:1' sf_internal_predicateOutput = In == true; *)

                    IF In THEN 
                        (* Transition: '<S49>:5' *)
                        is_c3_ChiefMaster := b_ChiefMaster_IN_Hold_h;
                        temporalCounter_i1(timerAction := 1, maxTime := 0);
                        (* Entry 'Hold': '<S49>:4' *)
                        (* '<S49>:4:2' Out = false *)
                        Out := FALSE;
                    ELSE 
                        (* '<S49>:1:2' Out = false *)
                        Out := FALSE;
                    END_IF;

                ELSE
                    (* During 'Hold': '<S49>:4' *)
                    (* '<S49>:8:1' sf_internal_predicateOutput = after(1,sec); *)
                    temporalCounter_i1(timerAction := 2, maxTime := 1000);

                    IF temporalCounter_i1.done THEN 
                        (* Transition: '<S49>:8' *)
                        is_c3_ChiefMaster := ChiefMaster_IN_Actual;
                        (* Entry 'Actual': '<S49>:7' *)
                        (* '<S49>:7:2' Out = In *)
                        Out := In;
                    ELSE 
                        (* '<S49>:9:1' sf_internal_predicateOutput = In==false; *)

                        IF  NOT In THEN 
                            (* Transition: '<S49>:9' *)
                            is_c3_ChiefMaster := ChiefMaster_IN_Default_e;
                            (* Entry 'Default': '<S49>:1' *)
                            (* '<S49>:1:2' Out = false *)
                            Out := FALSE;
                        ELSE 
                            (* '<S49>:4:2' Out = false *)
                            Out := FALSE;
                        END_IF;

                    END_IF;

            END_CASE;

        END_IF;

        (* End of Chart: '<S48>/Chart' *)
END_CASE;

END_FUNCTION_BLOCK

// Device/Application/InsulationMonitoringReq
FUNCTION_BLOCK InsulationMonitoringReq
VAR_INPUT
	ssMethodType: SINT;
	IT_boUDC_KL15_D: BOOL;
	IT_boUDC_KL15_C: BOOL;
	IT_boBMS_HV_ON_BB: BOOL;
	IT_u8BMS_BB_No_MaxVoltage: REAL;
	IT_u8BMS_BB_No_MinVoltage: REAL;
	IT_boBMS_SDError_BB1: BOOL;
	IT_boBMS_SDError_BB2: BOOL;
	IT_boBMS_SDError_BB3: BOOL;
	IT_boBMS_InsulationReadyOK_B1: BOOL;
	IT_boBMS_InsulationReadyOK_B2: BOOL;
	IT_boBMS_InsulationReadyOK_B3: BOOL;
	IT_boBMS_IMD_Active_BB1: BOOL;
	IT_boBMS_IMD_Active_BB2: BOOL;
	IT_boBMS_IMD_Active_BB3: BOOL;
	IT_boBMS_HV_REL_ON_BB1: BOOL;
	IT_boBMS_HV_REL_ON_BB2: BOOL;
	IT_boBMS_HV_REL_ON_BB3: BOOL;
	IT_sBMS_Batt1_Availability: LREAL;
	IT_sBMS_Batt2_Availability: LREAL;
	IT_sBMS_Batt3_Availability: LREAL;
	IT_boUDC_EV_IsolationMeasurementRequest: BOOL;
	FL_boSS_System_SD: BOOL;
	FL_boSS_System_ESD: BOOL;
END_VAR
VAR_OUTPUT
	FL_boREQ_IMD_ON_BB1: BOOL;
	FL_boREQ_IMD_ON_BB2: BOOL;
	FL_boREQ_IMD_ON_BB3: BOOL;
	FL_u8_IMD_State_BB1: USINT;
	FL_u8_IMD_State_BB2: USINT;
	FL_u8_IMD_State_BB3: USINT;
END_VAR
VAR
	i0_Chart_REQ_IMD_ON_BB1: Chart_REQ_IMD_ON_BB1;
	i0_Chart: Chart;
	i0_Chart_REQ_IMD_ON_BB2: Chart_REQ_IMD_ON_BB2;
	i1_Chart: Chart;
	i0_Chart_REQ_IMD_ON_BB3: Chart_REQ_IMD_ON_BB3;
	i2_Chart: Chart;
	rtb_OR_kt: BOOL;
	rtb_REQ_IMD_ON_k: BOOL;
END_VAR



CASE ssMethodType OF
    SS_INITIALIZE: 
        (* Constant: '<S48>/Constant9' *)
        i0_Chart_REQ_IMD_ON_BB1(ssMethodType := SS_INITIALIZE, ChargeMode := IT_boUDC_KL15_C, DriveMode := IT_boUDC_KL15_D, InsulationReadyOK := IT_boBMS_InsulationReadyOK_B1, MaxVtgBB := IT_u8BMS_BB_No_MaxVoltage, MinVtgBB := IT_u8BMS_BB_No_MinVoltage, SDError_BB := rtb_OR_kt, BattNo := BattBox1_No, HV_ON_BB := IT_boBMS_HV_ON_BB, IMD_Active_BB2 := IT_boBMS_IMD_Active_BB2, IMD_Active_BB3 := IT_boBMS_IMD_Active_BB3, IMD_Active_BB1 := IT_boBMS_IMD_Active_BB1, HV_REL_ON_BB := IT_boBMS_HV_REL_ON_BB1, BoxAvailable := IT_sBMS_Batt1_Availability, IsolationMeasurementRequest := IT_boUDC_EV_IsolationMeasurementRequest);
        rtb_REQ_IMD_ON_k := i0_Chart_REQ_IMD_ON_BB1.REQ_IMD_ON;
        FL_u8_IMD_State_BB1 := i0_Chart_REQ_IMD_ON_BB1.IMD_State;
        i0_Chart(ssMethodType := SS_INITIALIZE, In := rtb_REQ_IMD_ON_k);
        FL_boREQ_IMD_ON_BB1 := i0_Chart.Out;
        (* Constant: '<S48>/Constant1' *)
        i0_Chart_REQ_IMD_ON_BB2(ssMethodType := SS_INITIALIZE, ChargeMode := IT_boUDC_KL15_C, DriveMode := IT_boUDC_KL15_D, InsulationReadyOK := IT_boBMS_InsulationReadyOK_B2, MaxVtgBB := IT_u8BMS_BB_No_MaxVoltage, MinVtgBB := IT_u8BMS_BB_No_MinVoltage, SDError_BB := rtb_OR_kt, BattNo := BattBox2_No, HV_ON_BB := IT_boBMS_HV_ON_BB, IMD_Active_BB2 := IT_boBMS_IMD_Active_BB2, IMD_Active_BB3 := IT_boBMS_IMD_Active_BB3, IMD_Active_BB1 := IT_boBMS_IMD_Active_BB1, HV_REL_ON_BB := IT_boBMS_HV_REL_ON_BB2, BoxAvailable := IT_sBMS_Batt2_Availability, IsolationMeasurementRequest := IT_boUDC_EV_IsolationMeasurementRequest);
        rtb_REQ_IMD_ON_k := i0_Chart_REQ_IMD_ON_BB2.REQ_IMD_ON;
        FL_u8_IMD_State_BB2 := i0_Chart_REQ_IMD_ON_BB2.IMD_State;
        i1_Chart(ssMethodType := SS_INITIALIZE, In := rtb_REQ_IMD_ON_k);
        FL_boREQ_IMD_ON_BB2 := i1_Chart.Out;
        (* Constant: '<S48>/Constant2' *)
        i0_Chart_REQ_IMD_ON_BB3(ssMethodType := SS_INITIALIZE, ChargeMode := IT_boUDC_KL15_C, DriveMode := IT_boUDC_KL15_D, InsulationReadyOK := IT_boBMS_InsulationReadyOK_B3, MaxVtgBB := IT_u8BMS_BB_No_MaxVoltage, MinVtgBB := IT_u8BMS_BB_No_MinVoltage, SDError_BB := rtb_OR_kt, BattNo := BattBox3_No, HV_ON_BB := IT_boBMS_HV_ON_BB, IMD_Active_BB2 := IT_boBMS_IMD_Active_BB2, IMD_Active_BB3 := IT_boBMS_IMD_Active_BB3, IMD_Active_BB1 := IT_boBMS_IMD_Active_BB1, HV_REL_ON_BB := IT_boBMS_HV_REL_ON_BB3, BoxAvailable := IT_sBMS_Batt3_Availability, IsolationMeasurementRequest := IT_boUDC_EV_IsolationMeasurementRequest);
        rtb_REQ_IMD_ON_k := i0_Chart_REQ_IMD_ON_BB3.REQ_IMD_ON;
        FL_u8_IMD_State_BB3 := i0_Chart_REQ_IMD_ON_BB3.IMD_State;
        i2_Chart(ssMethodType := SS_INITIALIZE, In := rtb_REQ_IMD_ON_k);
        FL_boREQ_IMD_ON_BB3 := i2_Chart.Out;
    SS_OUTPUT: 
        (* Logic: '<S48>/OR' incorporates:
         *  Constant: '<S48>/Constant9' *)
        i0_Chart_REQ_IMD_ON_BB1(ssMethodType := SS_OUTPUT, ChargeMode := IT_boUDC_KL15_C, DriveMode := IT_boUDC_KL15_D, InsulationReadyOK := IT_boBMS_InsulationReadyOK_B1, MaxVtgBB := IT_u8BMS_BB_No_MaxVoltage, MinVtgBB := IT_u8BMS_BB_No_MinVoltage, SDError_BB := (IT_boBMS_SDError_BB1 OR FL_boSS_System_ESD) OR FL_boSS_System_SD, BattNo := BattBox1_No, HV_ON_BB := IT_boBMS_HV_ON_BB, IMD_Active_BB2 := IT_boBMS_IMD_Active_BB2, IMD_Active_BB3 := IT_boBMS_IMD_Active_BB3, IMD_Active_BB1 := IT_boBMS_IMD_Active_BB1, HV_REL_ON_BB := IT_boBMS_HV_REL_ON_BB1, BoxAvailable := IT_sBMS_Batt1_Availability, IsolationMeasurementRequest := IT_boUDC_EV_IsolationMeasurementRequest);
        rtb_REQ_IMD_ON_k := i0_Chart_REQ_IMD_ON_BB1.REQ_IMD_ON;
        FL_u8_IMD_State_BB1 := i0_Chart_REQ_IMD_ON_BB1.IMD_State;
        i0_Chart(ssMethodType := SS_OUTPUT, In := rtb_REQ_IMD_ON_k);
        FL_boREQ_IMD_ON_BB1 := i0_Chart.Out;
        (* Logic: '<S48>/OR1' incorporates:
         *  Constant: '<S48>/Constant1' *)
        i0_Chart_REQ_IMD_ON_BB2(ssMethodType := SS_OUTPUT, ChargeMode := IT_boUDC_KL15_C, DriveMode := IT_boUDC_KL15_D, InsulationReadyOK := IT_boBMS_InsulationReadyOK_B2, MaxVtgBB := IT_u8BMS_BB_No_MaxVoltage, MinVtgBB := IT_u8BMS_BB_No_MinVoltage, SDError_BB := (IT_boBMS_SDError_BB2 OR FL_boSS_System_SD) OR FL_boSS_System_ESD, BattNo := BattBox2_No, HV_ON_BB := IT_boBMS_HV_ON_BB, IMD_Active_BB2 := IT_boBMS_IMD_Active_BB2, IMD_Active_BB3 := IT_boBMS_IMD_Active_BB3, IMD_Active_BB1 := IT_boBMS_IMD_Active_BB1, HV_REL_ON_BB := IT_boBMS_HV_REL_ON_BB2, BoxAvailable := IT_sBMS_Batt2_Availability, IsolationMeasurementRequest := IT_boUDC_EV_IsolationMeasurementRequest);
        rtb_REQ_IMD_ON_k := i0_Chart_REQ_IMD_ON_BB2.REQ_IMD_ON;
        FL_u8_IMD_State_BB2 := i0_Chart_REQ_IMD_ON_BB2.IMD_State;
        i1_Chart(ssMethodType := SS_OUTPUT, In := rtb_REQ_IMD_ON_k);
        FL_boREQ_IMD_ON_BB2 := i1_Chart.Out;
        (* Logic: '<S48>/OR2' incorporates:
         *  Constant: '<S48>/Constant2' *)
        i0_Chart_REQ_IMD_ON_BB3(ssMethodType := SS_OUTPUT, ChargeMode := IT_boUDC_KL15_C, DriveMode := IT_boUDC_KL15_D, InsulationReadyOK := IT_boBMS_InsulationReadyOK_B3, MaxVtgBB := IT_u8BMS_BB_No_MaxVoltage, MinVtgBB := IT_u8BMS_BB_No_MinVoltage, SDError_BB := (IT_boBMS_SDError_BB3 OR FL_boSS_System_SD) OR FL_boSS_System_ESD, BattNo := BattBox3_No, HV_ON_BB := IT_boBMS_HV_ON_BB, IMD_Active_BB2 := IT_boBMS_IMD_Active_BB2, IMD_Active_BB3 := IT_boBMS_IMD_Active_BB3, IMD_Active_BB1 := IT_boBMS_IMD_Active_BB1, HV_REL_ON_BB := IT_boBMS_HV_REL_ON_BB3, BoxAvailable := IT_sBMS_Batt3_Availability, IsolationMeasurementRequest := IT_boUDC_EV_IsolationMeasurementRequest);
        rtb_REQ_IMD_ON_k := i0_Chart_REQ_IMD_ON_BB3.REQ_IMD_ON;
        FL_u8_IMD_State_BB3 := i0_Chart_REQ_IMD_ON_BB3.IMD_State;
        i2_Chart(ssMethodType := SS_OUTPUT, In := rtb_REQ_IMD_ON_k);
        FL_boREQ_IMD_ON_BB3 := i2_Chart.Out;
END_CASE;

END_FUNCTION_BLOCK

// Device/Application/Chart_REQ_IMD_ON_BB1
FUNCTION_BLOCK Chart_REQ_IMD_ON_BB1
VAR_INPUT
	ssMethodType: SINT;
	ChargeMode: BOOL;
	DriveMode: BOOL;
	InsulationReadyOK: BOOL;
	MaxVtgBB: REAL;
	MinVtgBB: REAL;
	SDError_BB: BOOL;
	BattNo: REAL;
	HV_ON_BB: BOOL;
	IMD_Active_BB2: BOOL;
	IMD_Active_BB3: BOOL;
	IMD_Active_BB1: BOOL;
	HV_REL_ON_BB: BOOL;
	BoxAvailable: LREAL;
	IsolationMeasurementRequest: BOOL;
END_VAR
VAR_OUTPUT
	REQ_IMD_ON: BOOL;
	IMD_State: USINT;
END_VAR
VAR
	is_c7_ChiefMaster: USINT;
	is_active_c7_ChiefMaster: USINT;
	is_DRIVE: USINT;
	is_CHARGE: USINT;
	tmp: BOOL;
END_VAR



CASE ssMethodType OF
    SS_INITIALIZE: 
        is_CHARGE := ChiefMaster_IN_NO_ACTIVE_CHILD_a;
        is_DRIVE := ChiefMaster_IN_NO_ACTIVE_CHILD_a;
        is_active_c7_ChiefMaster := 0;
        is_c7_ChiefMaster := ChiefMaster_IN_NO_ACTIVE_CHILD_a;
        REQ_IMD_ON := FALSE;
        IMD_State := 0;
    SS_OUTPUT: 
        (* Chart: '<S48>/Chart_REQ_IMD_ON_BB1' *)
        (* Gateway: ChiefMaster/Flow Logic/IMD Control/InsulationMonitoringReq/Chart_REQ_IMD_ON_BB1 *)
        (* During: ChiefMaster/Flow Logic/IMD Control/InsulationMonitoringReq/Chart_REQ_IMD_ON_BB1 *)

        IF is_active_c7_ChiefMaster = 0 THEN 
            (* Entry: ChiefMaster/Flow Logic/IMD Control/InsulationMonitoringReq/Chart_REQ_IMD_ON_BB1 *)
            is_active_c7_ChiefMaster := 1;
            (* Entry Internal: ChiefMaster/Flow Logic/IMD Control/InsulationMonitoringReq/Chart_REQ_IMD_ON_BB1 *)
            (* Transition: '<S52>:10' *)
            is_c7_ChiefMaster := ChiefMaster_IN_Default_fx;
            (* Entry 'Default': '<S52>:9' *)
            (* '<S52>:9:2' REQ_IMD_ON = false; *)
            REQ_IMD_ON := FALSE;
            (* '<S52>:9:3' IMD_State = uint8(0); *)
            IMD_State := 0;
        ELSE 

            CASE is_c7_ChiefMaster OF
                ChiefMaster_IN_CHARGE: 
                    (* During 'CHARGE': '<S52>:46' *)
                    (* '<S52>:21:1' sf_internal_predicateOutput = ((ChargeMode == false || DriveMode == true ||... *)
                    (* '<S52>:21:2'  SDError_BB == true || BoxAvailable==false) &&... *)
                    (* '<S52>:21:3' HV_REL_ON_BB == false); *)

                    IF (((( NOT ChargeMode) OR DriveMode) OR SDError_BB) OR (BoxAvailable = 0.0)) AND ( NOT HV_REL_ON_BB) THEN 
                        (* Transition: '<S52>:21' *)
                        (* Exit Internal 'CHARGE': '<S52>:46' *)
                        is_CHARGE := ChiefMaster_IN_NO_ACTIVE_CHILD_a;
                        is_c7_ChiefMaster := ChiefMaster_IN_Default_fx;
                        (* Entry 'Default': '<S52>:9' *)
                        (* '<S52>:9:2' REQ_IMD_ON = false; *)
                        REQ_IMD_ON := FALSE;
                        (* '<S52>:9:3' IMD_State = uint8(0); *)
                        IMD_State := 0;
                    ELSE 

                        CASE is_CHARGE OF
                            ChiefMaster_IN_CHARGE: 
                                (* During 'CHARGE': '<S52>:13' *)
                                (* '<S52>:32:1' sf_internal_predicateOutput = InsulationReadyOK == true &&... *)
                                (* '<S52>:32:2' MinVtgBB == BattNo &&... *)
                                (* '<S52>:32:3' HV_ON_BB == false; *)

                                IF (InsulationReadyOK AND (MinVtgBB = BattNo)) AND ( NOT HV_ON_BB) THEN 
                                    (* Transition: '<S52>:32' *)
                                    is_CHARGE := ChiefMaster_IN_IMD_ON;
                                    (* Entry 'IMD_ON': '<S52>:31' *)
                                    (* '<S52>:31:2' REQ_IMD_ON = true; *)
                                    REQ_IMD_ON := TRUE;
                                    (* '<S52>:31:3' IMD_State = uint8(5); *)
                                    IMD_State := 5;
                                ELSE 
                                    (* '<S52>:34:1' sf_internal_predicateOutput = (InsulationReadyOK == true && MinVtgBB ~=  BattNo) ||... *)
                                    (* '<S52>:34:2'  HV_ON_BB == true; *)

                                    IF (InsulationReadyOK AND (MinVtgBB <> BattNo)) OR HV_ON_BB THEN 
                                        (* Transition: '<S52>:34' *)
                                        is_CHARGE := ChiefMaster_IN_IMD_OFF;
                                        (* Entry 'IMD_OFF': '<S52>:33' *)
                                        (* '<S52>:33:2' REQ_IMD_ON = false; *)
                                        REQ_IMD_ON := FALSE;
                                        (* '<S52>:33:3' IMD_State = uint8(6); *)
                                        IMD_State := 6;
                                    ELSE 
                                        (* '<S52>:13:2' REQ_IMD_ON = true; *)
                                        REQ_IMD_ON := TRUE;
                                        (* '<S52>:13:3' IMD_State = uint8(4); *)
                                        IMD_State := 4;
                                    END_IF;

                                END_IF;

                            ChiefMaster_IN_IMD_OFF: 
                                (* During 'IMD_OFF': '<S52>:33' *)
                                (* '<S52>:75:1' sf_internal_predicateOutput = MinVtgBB == BattNo &&... *)
                                (* '<S52>:75:2' IMD_Active_BB1 == false &&... *)
                                (* '<S52>:75:3' IMD_Active_BB2 == false &&... *)
                                (* '<S52>:75:4' IMD_Active_BB3 == false &&... *)
                                (* '<S52>:75:5' IsolationMeasurementRequest == true; *)

                                IF ((((MinVtgBB = BattNo) AND ( NOT IMD_Active_BB1)) AND ( NOT IMD_Active_BB2)) AND ( NOT IMD_Active_BB3)) AND IsolationMeasurementRequest THEN 
                                    (* Transition: '<S52>:75' *)
                                    is_CHARGE := ChiefMaster_IN_IMD_ON;
                                    (* Entry 'IMD_ON': '<S52>:31' *)
                                    (* '<S52>:31:2' REQ_IMD_ON = true; *)
                                    REQ_IMD_ON := TRUE;
                                    (* '<S52>:31:3' IMD_State = uint8(5); *)
                                    IMD_State := 5;
                                ELSE 
                                    (* '<S52>:33:2' REQ_IMD_ON = false; *)
                                    REQ_IMD_ON := FALSE;
                                    (* '<S52>:33:3' IMD_State = uint8(6); *)
                                    IMD_State := 6;
                                END_IF;

                            ELSE
                                (* During 'IMD_ON': '<S52>:31' *)
                                (* '<S52>:87:1' sf_internal_predicateOutput = HV_ON_BB == true &&... *)
                                (* '<S52>:87:2' IsolationMeasurementRequest == false; *)

                                IF HV_ON_BB AND ( NOT IsolationMeasurementRequest) THEN 
                                    (* Transition: '<S52>:87' *)
                                    is_CHARGE := ChiefMaster_IN_IMD_OFF;
                                    (* Entry 'IMD_OFF': '<S52>:33' *)
                                    (* '<S52>:33:2' REQ_IMD_ON = false; *)
                                    REQ_IMD_ON := FALSE;
                                    (* '<S52>:33:3' IMD_State = uint8(6); *)
                                    IMD_State := 6;
                                ELSE 
                                    (* '<S52>:31:2' REQ_IMD_ON = true; *)
                                    REQ_IMD_ON := TRUE;
                                    (* '<S52>:31:3' IMD_State = uint8(5); *)
                                    IMD_State := 5;
                                END_IF;

                        END_CASE;

                    END_IF;

                ChiefMaster_IN_DRIVE: 
                    (* During 'DRIVE': '<S52>:62' *)
                    (* '<S52>:27:1' sf_internal_predicateOutput = ((DriveMode == false || ChargeMode == true ||... *)
                    (* '<S52>:27:2' SDError_BB == true || BoxAvailable==false) &&... *)
                    (* '<S52>:27:3' HV_REL_ON_BB == false); *)

                    IF (((( NOT DriveMode) OR ChargeMode) OR SDError_BB) OR (BoxAvailable = 0.0)) AND ( NOT HV_REL_ON_BB) THEN 
                        (* Transition: '<S52>:27' *)
                        (* Exit Internal 'DRIVE': '<S52>:62' *)
                        is_DRIVE := ChiefMaster_IN_NO_ACTIVE_CHILD_a;
                        is_c7_ChiefMaster := ChiefMaster_IN_Default_fx;
                        (* Entry 'Default': '<S52>:9' *)
                        (* '<S52>:9:2' REQ_IMD_ON = false; *)
                        REQ_IMD_ON := FALSE;
                        (* '<S52>:9:3' IMD_State = uint8(0); *)
                        IMD_State := 0;
                    ELSE 

                        CASE is_DRIVE OF
                            ChiefMaster_IN_DRIVE_d: 
                                (* During 'DRIVE': '<S52>:63' *)
                                (* '<S52>:67:1' sf_internal_predicateOutput = InsulationReadyOK == true &&... *)
                                (* '<S52>:67:2' MaxVtgBB == BattNo &&... *)
                                (* '<S52>:67:3' HV_ON_BB == false; *)

                                IF (InsulationReadyOK AND (MaxVtgBB = BattNo)) AND ( NOT HV_ON_BB) THEN 
                                    (* Transition: '<S52>:67' *)
                                    is_DRIVE := ChiefMaster_IN_IMD_ON;
                                    (* Entry 'IMD_ON': '<S52>:64' *)
                                    (* '<S52>:64:2' REQ_IMD_ON = true; *)
                                    REQ_IMD_ON := TRUE;
                                    (* '<S52>:64:3' IMD_State = uint8(2); *)
                                    IMD_State := 2;
                                ELSE 
                                    (* '<S52>:68:1' sf_internal_predicateOutput = (InsulationReadyOK == true && MaxVtgBB ~=  BattNo)  ||... *)
                                    (* '<S52>:68:2' HV_ON_BB == true; *)

                                    IF (InsulationReadyOK AND (MaxVtgBB <> BattNo)) OR HV_ON_BB THEN 
                                        (* Transition: '<S52>:68' *)
                                        is_DRIVE := ChiefMaster_IN_IMD_OFF;
                                        (* Entry 'IMD_OFF': '<S52>:65' *)
                                        (* '<S52>:65:2' REQ_IMD_ON = false; *)
                                        REQ_IMD_ON := FALSE;
                                        (* '<S52>:65:3' IMD_State = uint8(3); *)
                                        IMD_State := 3;
                                    ELSE 
                                        (* '<S52>:63:2' REQ_IMD_ON = true; *)
                                        REQ_IMD_ON := TRUE;
                                        (* '<S52>:63:3' IMD_State = uint8(1); *)
                                        IMD_State := 1;
                                    END_IF;

                                END_IF;

                            ChiefMaster_IN_IMD_OFF: 
                                (* During 'IMD_OFF': '<S52>:65' *)
                                (* '<S52>:77:1' sf_internal_predicateOutput = MaxVtgBB == BattNo &&... *)
                                (* '<S52>:77:2' IMD_Active_BB1 == false &&... *)
                                (* '<S52>:77:3' IMD_Active_BB2 == false &&... *)
                                (* '<S52>:77:4' IMD_Active_BB3 == false &&... *)
                                (* '<S52>:77:5' IsolationMeasurementRequest == true; *)

                                IF ((((MaxVtgBB = BattNo) AND ( NOT IMD_Active_BB1)) AND ( NOT IMD_Active_BB2)) AND ( NOT IMD_Active_BB3)) AND IsolationMeasurementRequest THEN 
                                    (* Transition: '<S52>:77' *)
                                    is_DRIVE := ChiefMaster_IN_IMD_ON;
                                    (* Entry 'IMD_ON': '<S52>:64' *)
                                    (* '<S52>:64:2' REQ_IMD_ON = true; *)
                                    REQ_IMD_ON := TRUE;
                                    (* '<S52>:64:3' IMD_State = uint8(2); *)
                                    IMD_State := 2;
                                ELSE 
                                    (* '<S52>:65:2' REQ_IMD_ON = false; *)
                                    REQ_IMD_ON := FALSE;
                                    (* '<S52>:65:3' IMD_State = uint8(3); *)
                                    IMD_State := 3;
                                END_IF;

                            ELSE
                                (* During 'IMD_ON': '<S52>:64' *)
                                (* '<S52>:88:1' sf_internal_predicateOutput = HV_ON_BB == true &&... *)
                                (* '<S52>:88:2' IsolationMeasurementRequest == false; *)

                                IF HV_ON_BB AND ( NOT IsolationMeasurementRequest) THEN 
                                    (* Transition: '<S52>:88' *)
                                    is_DRIVE := ChiefMaster_IN_IMD_OFF;
                                    (* Entry 'IMD_OFF': '<S52>:65' *)
                                    (* '<S52>:65:2' REQ_IMD_ON = false; *)
                                    REQ_IMD_ON := FALSE;
                                    (* '<S52>:65:3' IMD_State = uint8(3); *)
                                    IMD_State := 3;
                                ELSE 
                                    (* '<S52>:64:2' REQ_IMD_ON = true; *)
                                    REQ_IMD_ON := TRUE;
                                    (* '<S52>:64:3' IMD_State = uint8(2); *)
                                    IMD_State := 2;
                                END_IF;

                        END_CASE;

                    END_IF;

                ELSE
                    (* During 'Default': '<S52>:9' *)
                    (* '<S52>:14:1' sf_internal_predicateOutput = ChargeMode == true && DriveMode == false &&... *)
                    (* '<S52>:14:2'  SDError_BB == false && BoxAvailable==true; *)
                    tmp :=  NOT SDError_BB;

                    IF ((ChargeMode AND ( NOT DriveMode)) AND tmp) AND (BoxAvailable = 1.0) THEN 
                        (* Transition: '<S52>:14' *)
                        is_c7_ChiefMaster := ChiefMaster_IN_CHARGE;
                        (* Entry Internal 'CHARGE': '<S52>:46' *)
                        (* Transition: '<S52>:47' *)
                        is_CHARGE := ChiefMaster_IN_CHARGE;
                        (* Entry 'CHARGE': '<S52>:13' *)
                        (* '<S52>:13:2' REQ_IMD_ON = true; *)
                        REQ_IMD_ON := TRUE;
                        (* '<S52>:13:3' IMD_State = uint8(4); *)
                        IMD_State := 4;
                    ELSE 
                        (* '<S52>:18:1' sf_internal_predicateOutput = DriveMode == true && ChargeMode == false &&... *)
                        (* '<S52>:18:2'  SDError_BB == false && BoxAvailable==true; *)

                        IF ((DriveMode AND ( NOT ChargeMode)) AND tmp) AND (BoxAvailable = 1.0) THEN 
                            (* Transition: '<S52>:18' *)
                            is_c7_ChiefMaster := ChiefMaster_IN_DRIVE;
                            (* Entry Internal 'DRIVE': '<S52>:62' *)
                            (* Transition: '<S52>:66' *)
                            is_DRIVE := ChiefMaster_IN_DRIVE_d;
                            (* Entry 'DRIVE': '<S52>:63' *)
                            (* '<S52>:63:2' REQ_IMD_ON = true; *)
                            REQ_IMD_ON := TRUE;
                            (* '<S52>:63:3' IMD_State = uint8(1); *)
                            IMD_State := 1;
                        ELSE 
                            (* '<S52>:9:2' REQ_IMD_ON = false; *)
                            REQ_IMD_ON := FALSE;
                            (* '<S52>:9:3' IMD_State = uint8(0); *)
                            IMD_State := 0;
                        END_IF;

                    END_IF;

            END_CASE;

        END_IF;

        (* End of Chart: '<S48>/Chart_REQ_IMD_ON_BB1' *)
END_CASE;

END_FUNCTION_BLOCK

// Device/Application/Chart_REQ_IMD_ON_BB2
FUNCTION_BLOCK Chart_REQ_IMD_ON_BB2
VAR_INPUT
	ssMethodType: SINT;
	ChargeMode: BOOL;
	DriveMode: BOOL;
	InsulationReadyOK: BOOL;
	MaxVtgBB: REAL;
	MinVtgBB: REAL;
	SDError_BB: BOOL;
	BattNo: REAL;
	HV_ON_BB: BOOL;
	IMD_Active_BB2: BOOL;
	IMD_Active_BB3: BOOL;
	IMD_Active_BB1: BOOL;
	HV_REL_ON_BB: BOOL;
	BoxAvailable: LREAL;
	IsolationMeasurementRequest: BOOL;
END_VAR
VAR_OUTPUT
	REQ_IMD_ON: BOOL;
	IMD_State: USINT;
END_VAR
VAR
	is_c66_ChiefMaster: USINT;
	is_active_c66_ChiefMaster: USINT;
	is_DRIVE: USINT;
	is_CHARGE: USINT;
	tmp: BOOL;
END_VAR



CASE ssMethodType OF
    SS_INITIALIZE: 
        is_CHARGE := ChiefMaster_IN_NO_ACTIVE_CHILD_jz;
        is_DRIVE := ChiefMaster_IN_NO_ACTIVE_CHILD_jz;
        is_active_c66_ChiefMaster := 0;
        is_c66_ChiefMaster := ChiefMaster_IN_NO_ACTIVE_CHILD_jz;
        REQ_IMD_ON := FALSE;
        IMD_State := 0;
    SS_OUTPUT: 
        (* Chart: '<S48>/Chart_REQ_IMD_ON_BB2' *)
        (* Gateway: ChiefMaster/Flow Logic/IMD Control/InsulationMonitoringReq/Chart_REQ_IMD_ON_BB2 *)
        (* During: ChiefMaster/Flow Logic/IMD Control/InsulationMonitoringReq/Chart_REQ_IMD_ON_BB2 *)

        IF is_active_c66_ChiefMaster = 0 THEN 
            (* Entry: ChiefMaster/Flow Logic/IMD Control/InsulationMonitoringReq/Chart_REQ_IMD_ON_BB2 *)
            is_active_c66_ChiefMaster := 1;
            (* Entry Internal: ChiefMaster/Flow Logic/IMD Control/InsulationMonitoringReq/Chart_REQ_IMD_ON_BB2 *)
            (* Transition: '<S53>:10' *)
            is_c66_ChiefMaster := ChiefMaster_IN_Default_d;
            (* Entry 'Default': '<S53>:9' *)
            (* '<S53>:9:2' REQ_IMD_ON = false; *)
            REQ_IMD_ON := FALSE;
            (* '<S53>:9:3' IMD_State = uint8(0); *)
            IMD_State := 0;
        ELSE 

            CASE is_c66_ChiefMaster OF
                ChiefMaster_IN_CHARGE_c: 
                    (* During 'CHARGE': '<S53>:46' *)
                    (* '<S53>:21:1' sf_internal_predicateOutput = ((ChargeMode == false || DriveMode == true ||... *)
                    (* '<S53>:21:2'  SDError_BB == true || BoxAvailable==false) &&... *)
                    (* '<S53>:21:3' HV_REL_ON_BB == false); *)

